(* CODESYS project Test Project V2.project

Project tree, tasks and I/O mapping:
  Device : CODESYS Control Win V3, 3S - Smart Software Solutions GmbH, order no. 305021, version 3.5.7.10
    application Application
      libraries: Standard, * (System)
      task MainTask (cyclic, interval t#500ms, priority 10) calls PLC_PRG
      program PLC_PRG [ST]
  libraries: Standard, 3.5.7.0 (System); SystemTask, 1.3.5.0 (SEL)
  Program/
    Global_Variables/
      global variables Generator_GLV
      global variables Meter_GLV
      global variables Reactive_Bank_GLV
      global variables Run_Time_GLV
    Core Function Blocks/
      function block Circuit_Master [ST]
      function block Power_Control [ST]
      function block Reactive_Control [ST]
      function block Reactive_Bank_Control [ST]
      program Run_Time_Header [ST]
      function block Cap_Bank_Control [ST]
      function block Volt_Var [ST]
      function block Voltage_Control [ST]
    Functions/
      function block PI_Controller [ST]
      function Linearize [ST]
      function PF_to_KVAr [ST]
      Generator_Functions/
        function Generic_Trigger [ST]
        function block Generator_Volt_Var [ST]
        function block Generator_Power_Ramp [ST]
    Interface Blocks/
      function block Reactive_Bank_Interface [ST]
      function block Generic_Generator [ST]
      function block AE_1000NX [ST]
      function block AE_500NX [ST]
      function block SMA_800CP [ST]
      function block SMA_2200CP [ST]
      function block TMEIC_PVL1833 [ST]
      function block Schneider_ConextCore_XC [ST]
      function block SG_1000MX [ST]
*)

// Program/Global_Variables/Generator_GLV
VAR_GLOBAL
	
	// Boolean Reads
	POIV2_Generator_Offline 			: ARRAY[0..99] OF BOOL := [100(0)];
	POIV2_Generator_Fault 				: ARRAY[0..99] OF BOOL := [100(0)];
	POIV2_Generator_DNR					: ARRAY[0..99] OF BOOL := [100(0)];	
	POIV2_Generator_Volt_Var_Protection	: ARRAY[0..99] OF BOOL := [100(0)];
	
	// Boolean Writes
	POIV2_Generator_ON_OFF_CMD 			: ARRAY[0..99] OF BOOL := [100(1)];
	
	//Analog Reads
	POIV2_Circuit_Number 				: ARRAY[0..99] OF REAL := [100(-1)];
	POIV2_Block_Number 					: ARRAY[0..99] OF REAL := [100(-1)];
	POIV2_Generator_Number 				: ARRAY[0..99] OF REAL := [100(-1)];
	POIV2_Generator_KW 					: ARRAY[0..99] OF REAL := [100(1)];
	POIV2_Generator_KVAr 				: ARRAY[0..99] OF REAL := [100(1)];
	POIV2_Generator_PF 					: ARRAY[0..99] OF REAL := [100(1)];
	POIV2_Generator_Max_KW 				: ARRAY[0..99] OF REAL := [100(1)];
	POIV2_Generator_Max_KVAr 			: ARRAY[0..99] OF REAL := [100(1)];
		
	//Analog Writes
	POIV2_Generator_Power_Mode_SP 		: ARRAY[0..99] OF REAL := [100(0)];
	POIV2_Generator_Reactive_Mode_SP 	: ARRAY[0..99] OF REAL := [100(0)];
	POIV2_Generator_Volt_Var_Mode_SP	: ARRAY[0..99] OF REAL := [100(0)];
	POIV2_Generator_PF_SP 				: ARRAY[0..99] OF REAL := [100(1)];
	POIV2_Generator_PF_Ramp_SP 			: ARRAY[0..99] OF REAL := [100(0)];
	POIV2_Generator_KW_Percent_SP		: ARRAY[0..99] OF REAL := [100(100)];
	POIV2_Generator_KW_Ramp_SP 			: ARRAY[0..99] OF REAL := [100(0)];
	POIV2_Generator_KVAr_SP 			: ARRAY[0..99] OF REAL := [100(100)];
	POIV2_Generator_KVAr_Ramp_SP 		: ARRAY[0..99] OF REAL := [100(0)];
	
	//Calculated Analog Reads
	POIV2_Generator_Calculated_KW_Percent_SP 	: ARRAY[0..99] OF REAL := [100(100)];	//Sends feedback from setpoint ramping
	
	POIV2_Power_Redistribution_Mode				: ARRAY[0..99] OF INT := [100(0)]; 
	POIV2_Generator_Overhead_Percent			: ARRAY[0..99] OF REAL := [100(1)];	//Used in Power_Redistribution_Mode
	POIV2_Generator_Surplus_Percent		 		: ARRAY[0..99] OF REAL := [100(1)];	//Used in Power_Redistribution_Mode
	
END_VAR

// Program/Global_Variables/Meter_GLV
VAR_GLOBAL
	// Boolean Reads
	POIV2_Circuit_Breaker_State 	: ARRAY[0..9] OF BOOL := [10(0)];
	POIV2_Circuit_Meter_Offline 	: ARRAY[0..9] OF BOOL := [10(1)];
	                                                          
	//Analog Reads                                            
	POIV2_Circuit_Meter_KW 			: ARRAY[0..9] OF REAL := [10(0)];
	POIV2_Circuit_Meter_KVAr 		: ARRAY[0..9] OF REAL := [10(0)];
	POIV2_Circuit_Meter_PF 			: ARRAY[0..9] OF REAL := [10(1)];
	POIV2_Circuit_Meter_Frequency 	: ARRAY[0..9] OF REAL := [10(0)];
	POIV2_Circuit_Meter_KV 			: ARRAY[0..9] OF REAL := [10(0)];
END_VAR

// Program/Global_Variables/Reactive_Bank_GLV
VAR_GLOBAL


	//Boolean Reads
	POIV2_Cap_Bank_Offline 				: ARRAY[0..9] OF BOOL := [10(0)];
	POIV2_Cap_Bank_Fault 				: ARRAY[0..9] OF BOOL := [10(0)];
	POIV2_Cap_Bank_On	 				: ARRAY[0..9] OF BOOL := [10(0)];
	POIV2_Cap_Bank_Discharging			: ARRAY[0..9] OF BOOL := [10(0)];
	POIV2_Cap_Bank_Switch_Count_Reached	: ARRAY[0..9] OF BOOL := [10(0)];
	
	//Boolean Writes
	POIV2_Cap_Bank_ON_OFF_CMD 			: ARRAY[0..9] OF BOOL := [10(0)];
	POIV2_Cap_Bank_Reset				: ARRAY[0..9] OF BOOL := [10(0)];
	
	
	//Analog Reads
	Reactive_Bank_DNR_Count 			: ARRAY[0..9] OF INT := [10(-1)]; 
	POIV2_Cap_Bank_Circuit_Number 		: ARRAY[0..9] OF INT := [10(-1)];
	POIV2_Cap_Bank_Normalized_KVAr 		: ARRAY[0..9] OF REAL := [10(1000000.0)];
	POIV2_Cap_Bank_Operations_Count 	: ARRAY[0..9] OF REAL ;
	
	
	
	
	
	//Boolean Reads
	POIV2_Reactor_Bank_Offline 				: ARRAY[0..9] OF BOOL := [10(1)];
	POIV2_Reactor_Bank_Fault 				: ARRAY[0..9] OF BOOL := [10(1)];
	POIV2_Reactor_Bank_On	 				: ARRAY[0..9] OF BOOL := [10(0)];
	POIV2_Reactor_Bank_Discharging			: ARRAY[0..9] OF BOOL := [10(0)];
	POIV2_Reactor_Bank_Switch_Count_Reached	: ARRAY[0..9] OF BOOL := [10(0)];
	
	//Boolean Writes
	POIV2_Reactor_Bank_ON_OFF_CMD 			: ARRAY[0..9] OF BOOL := [10(0)];
	POIV2_Reactor_Bank_Reset				: ARRAY[0..9] OF BOOL := [10(0)];
	
	//Analog Reads
	POIV2_Reactor_Bank_Circuit_Number 		: ARRAY[0..9] OF INT := [10(-1)];
	POIV2_Reactor_Bank_Normalized_KVAr 		: ARRAY[0..9] OF REAL := [10(-1000000.0)];
	POIV2_Reactor_Bank_Operations_Count 	: ARRAY[0..9] OF REAL ;
END_VAR

// Program/Global_Variables/Run_Time_GLV
VAR_GLOBAL
	
	//Internal
	
	//{ attribute 'hide' }
	POIV2_Generator_Count	: INT := -1;
	//{ attribute 'hide' }
	POIV2_Reactive_Bank_Count	: INT := -1;
	
	
	
	//{ attribute 'hide' }
	Master_Power_Control_License : BOOL := TRUE;
	//{ attribute 'hide' }
	Master_Reactive_Control_License : BOOL := TRUE;
	
	Power_Control_Disable		: ARRAY[0..10] OF BOOL := [10(1)];
	Reactive_Control_Disable	: ARRAY[0..10] OF BOOL := [10(1)];
	Reactive_Bank_Disable	 	: ARRAY[0..10] OF BOOL := [10(1)];
	Volt_Var_Disable			: ARRAY[0..10] OF BOOL := [10(1)];
	Freq_Watt_Disable			: ARRAY[0..10] OF BOOL := [10(1)]; 
	Voltage_Controller_Disable  : ARRAY[0..10] OF BOOL := [10(1)];
	
	
	//Controller States
	//Controller_States	: ARRAY[0..10] OF BOOL := [10(0)];
	
	//Controller Alarms
	
	
END_VAR

// Device/Application/PLC_PRG
PROGRAM PLC_PRG
VAR 
	Circuit_1_Master : Circuit_Master;
	Circuit_Power_Control : Power_Control;
	Circuit_1_Reactive_Control : Reactive_Control;
	Circuit1_Cap_Control : Cap_Bank_Control;
	
	Circuit1_Circuit_Number			: INT	;
	Circuit1_Breaker_State 			: BOOL	;
	Circuit1_Meter_Offline 			: BOOL	;
	
	Power_Mode : INT;
	counter : INT;
END_VAR

Run_Time_Header();

Circuit_1_Master(
	Circuit_Number	:= 	0,      
	Breaker_State 	:= 	0,      
	Meter_Offline 	:= 	0);   
	
	
	Circuit_Power_Control(
	Circuit_Number:= 0, 
	Disable:= FALSE, 
	Control_Mode:= Power_Mode, 
	Circuit_KW_SP:= 8000, 
	Line_Loss_Modifier:= 1, 
	Circuit_Ramp_Up_Rate:= 60, 
	Circuit_Ramp_Down_Rate:= 60, 
	Generator_Ramp_Rate:= 60, 
	KP:= 0.01, 
	KI:= 1, 
	Run_Cycle:= T#1S);
	
	
	

	Circuit1_Cap_Control(
	Circuit_Number:= 0, 
	Disable:= FALSE, 
	Reset:= FALSE);
	
	
	
	
	
	
	
	
	
	
	
//Test Variables
Circuit_1_Master.Meter_KW 	:= 	Circuit_1_Master.Generators_Gross_KW / 1.05;
Circuit_1_Master.Meter_KVAr := 	Circuit_1_Master.Generators_Gross_KW - 1500 + Circuit1_Cap_Control.Current_Cap_KVAr;
Circuit_1_Master.Meter_PF 	:= LREAL_TO_REAL(Circuit_1_Master.Meter_KW/EXPT(EXPT(Circuit_1_Master.Meter_KW,2)+EXPT(Circuit_1_Master.Meter_KVAr,2),0.5));

FOR counter := 0 TO 99 BY 1 DO
	Generator_GLV.POIV2_Generator_KW[counter] := Generator_GLV.POIV2_Generator_KW_Percent_SP[counter] * 10;
	Generator_GLV.POIV2_Generator_Max_KW[counter] := 1000;
	Generator_GLV.POIV2_Generator_Max_KVAr[counter] := 1000;
	Generator_GLV.POIV2_Generator_KVAr[counter] := linearize(Generator_GLV.POIV2_Generator_PF_SP[counter]) * 1000;
END_FOR

FOR counter := 0 TO 9 BY 1 DO
	Reactive_Bank_GLV.POIV2_Cap_Bank_On[counter] := Reactive_Bank_GLV.POIV2_Cap_Bank_ON_OFF_CMD[counter];
END_FOR

END_PROGRAM

// Program/Core Function Blocks/Run_Time_Header
PROGRAM Run_Time_Header
VAR
	{ attribute 'hide' }
	counter : INT;
	{ attribute 'hide' }
	model : STRING;
	{ attribute 'hide' }
	number : INT;
	{ attribute 'hide' }
	A : BOOL;
	{ attribute 'hide' }
	B : BOOL;
	{ attribute 'hide' }
	C : BOOL;
	{ attribute 'hide' }
	D : BOOL;
END_VAR


Run_Time_GLV.POIV2_Generator_Count 		:= 0;
Run_Time_GLV.POIV2_Reactive_Bank_Count 	:= 0;


Run_Time_GLV.Master_Power_Control_License 		:= TRUE;
Run_Time_GLV.Master_Reactive_Control_License 	:= TRUE;


GET_MOT(Model);
A := FALSE;
B := FALSE;
C := FALSE;
D := FALSE;
Number := 0;
IF(LEFT(Right(Model,2),1) = 'S')THEN
	Number  := STRING_TO_INT(CONCAT('16#',(Right(Model,1))));
	IF(Number > 15)THEN
		Number := 0;
	END_IF
	IF(Number >= 8)THEN
		D := TRUE;
		Number := Number -8;
	END_IF 
	IF(Number >= 4)THEN
		C := TRUE;
		Number := Number - 4;
	END_IF
	IF(Number >= 2)THEN
		B := TRUE;
		Number := Number - 2;
	END_IF
	IF(Number = 1)THEN
		A := TRUE;
		Number := Number - 1;
	END_IF
ELSIF(LEFT(Right(Model,4),2) = 'G1')THEN
	A := TRUE;
	B := TRUE;
ELSE
	A := FALSE;
	B := FALSE;
	C := FALSE;
	D := FALSE;
END_IF


//Run_Time_GLV.Master_Power_Control_License 		:= A;
//Run_Time_GLV.Master_Reactive_Control_License 	:= B;

END_PROGRAM

// Program/Functions/Linearize
FUNCTION Linearize : REAL
VAR_INPUT
	PF : REAL;
END_VAR

IF(PF >= 0)THEN
	Linearize := (1-PF);
ELSE
	Linearize := -1*(1+PF);
END_IF

END_FUNCTION

// Program/Core Function Blocks/Circuit_Master
FUNCTION_BLOCK Circuit_Master
VAR_INPUT
	Circuit_Number			: INT	:= 1;
	Breaker_State 			: BOOL	:= FALSE;
	Meter_Offline 			: BOOL	:= TRUE;
	Meter_KW				: REAL	:= 0;
	Meter_KVAr				: REAL	:= 0;
	Meter_PF				: REAL	:= 1;
	Meter_KV				: REAL	:= 0;
	Meter_Frequency			: REAL	:= 0;
	Generator_Power_Mode	: INT	:= 0; //0 = no power control || 1 = Active Power Limit Control
	Generator_Reactive_Mode	: INT	:= 0; //0 = unity power || 1 = KVAr Control || 2 = Power Factor Control
	Generator_Volt_Var_Mode : INT 	:= 0; //0 = Generators produce VArs even if they trip off to over/under voltage ||1 = Generators produce VArs unill the voltage is too high/low on the output terminals and reduces VArs
END_VAR
VAR_OUTPUT
	Curtail_Licenced					: BOOL;
	PF_Licenced							: BOOL;
	POI_Status 							: INT;
	POI_Alarms 							: INT;
	Generators_In_Control_Loop			: INT;
	Generators_Offline 					: INT;
	Generators_Faulted 					: INT;
	Generators_In_Volt_Var_Protection	: INT;
	Generators_DNR						: INT;
	Generators_Gross_KW 				: REAL;
	Generators_Gross_KVAr 				: REAL;

END_VAR
VAR
	{ attribute 'hide' }
	counter : INT;
END_VAR



// Variable Meter_GLV Writes 			
Meter_GLV.POIV2_Circuit_Breaker_State[Circuit_Number] 	:= Breaker_State; 	
Meter_GLV.POIV2_Circuit_Meter_Offline[Circuit_Number] 	:= Meter_Offline; 	 	
Meter_GLV.POIV2_Circuit_Meter_KW[Circuit_Number] 		:= Meter_KW;
Meter_GLV.POIV2_Circuit_Meter_KVAr[Circuit_Number] 		:= Meter_KVAr;
Meter_GLV.POIV2_Circuit_Meter_PF[Circuit_Number] 		:= Meter_PF;
Meter_GLV.POIV2_Circuit_Meter_Frequency[Circuit_Number] := Meter_Frequency;
Meter_GLV.POIV2_Circuit_Meter_KV[Circuit_Number] 		:= Meter_KV;



// Reset values
Generators_In_Control_Loop	:= 0;
Generators_Offline 			:= 0; 
Generators_Faulted 			:= 0; 
Generators_DNR 				:= 0;
Generators_Gross_KW 		:= 0; 
Generators_Gross_KVAr		:= 0; 

FOR counter := 0 TO 99 BY 1 DO
	IF(Generator_GLV.POIV2_Circuit_Number[counter] = Circuit_Number)THEN
		
		// Variable Generator_GLV Reads
		IF((Generator_GLV.POIV2_Generator_Offline[counter] = 0) AND (Generator_GLV.POIV2_Generator_Fault[counter] = 0))THEN
			Generators_In_Control_Loop 	:= Generators_In_Control_Loop + 1;
		END_IF
		
		Generators_Offline 			:= BOOL_TO_INT(Generator_GLV.POIV2_Generator_Offline[counter])	+ Generators_Offline;
		Generators_Faulted 			:= BOOL_TO_INT(Generator_GLV.POIV2_Generator_Fault[counter]) 	+ Generators_Faulted;
		Generators_DNR 				:= BOOL_TO_INT(Generator_GLV.POIV2_Generator_DNR[counter]) 		+ Generators_DNR;
		Generators_Gross_KW 		:= Generator_GLV.POIV2_Generator_KW[counter] 		+ Generators_Gross_KW;
		Generators_Gross_KVAr		:= Generator_GLV.POIV2_Generator_KVAr[counter] 		+ Generators_Gross_KVAr;
		// Variable Generator_GLV Writes
		Generator_GLV.POIV2_Generator_Power_Mode_SP[counter] 	:= Generator_Power_Mode;
		Generator_GLV.POIV2_Generator_Reactive_Mode_SP[counter] := Generator_Reactive_Mode;
		Generator_GLV.POIV2_Generator_Volt_Var_Mode_SP[counter] := Generator_Volt_Var_Mode;
	END_IF
END_FOR

END_FUNCTION_BLOCK

// Program/Core Function Blocks/Power_Control
FUNCTION_BLOCK Power_Control
VAR_INPUT
	Circuit_Number 			: INT	:= 1;	//Circuit Number for control
	Disable					: BOOL	:= FALSE;	//TRUE fully disables this controller || FALSE enables the controller
	Control_Mode			: INT	:= 0;	//0=Fixed Rate || 1=Dynamic Balance Conservative || 2=Dynamic Balance Moderate || 3=Dynamic Balance Aggressive || 4=PI Control
	Power_Redistribution_Mode: INT	:= 0;   //0=Power Controller sends the same command to all of the Inverters || 1=Inverters Reroute power based on avaliablity  ||Note: Speed Dependant on the feedback time of the end device
	Max_Circuit_KW 			: REAL 	:= 10000; //Maximum AC Power
	Circuit_KW_SP			: REAL	:= 1500;	//KW Circuit Setpoint
	Line_Loss_Modifier		: REAL 	:= 1.02; //
	Circuit_Ramp_Up_Rate	: REAL	:= 10; //KW Per Minute
	Circuit_Ramp_Down_Rate	: REAL	:= 10; //KW Per Minute
	Generator_Ramp_Rate		: REAL	:= 10; //KW Per Minute
	Deadband				: REAL 	:= 10;//Used in PI Control
	KP						: REAL	:= 0.01;//Tuning Parameter for the proportional constant
	KI						: REAL	:= 0.1;//Tuning Parameter for the integral constant
	Run_Cycle				: TIME	:= T#1S;
END_VAR
VAR
	PI_Control : PI_Controller;
	Run_Timer 	: TON;
	Jump_Timer	: TON;
	Offline_Generator_ON_Timer : TON;
	Offline_Generator_OFF_Timer : TON;
	
	counter : INT;
	
	Generators_Count 	: INT;
	Generators_Offline 	: INT;
	Generators_Faulted 	: INT;
	Generators_Gross_KW : REAL;
	Generators_Max_KW 	: REAL;
	Generators_In_Control_Loop : INT;
	Generators_Unknown_Offline_KW 	: REAL;
	Generators_Faulted_KW : REAL;
	
	Final_Circuit_KW_SP : REAL;
	Post_Ramp_Circuit_KW_SP : REAL;
	Offline_Generators_Estimated_Faulted : INT;
	Offline_Generators_KW_Correction : REAL;
	Old_Generators_Offline : INT;
	
	OLD_Generator_KW_Percent : REAL := 100;
	
	OLD_Circuit_KW_SP : REAL := 1000000;
	Ramp_Down_Value : REAL;
	Ramp_Up_Value : REAL;
	
	PI_Control_EN : BOOL := FALSE;
	PI_Control_Offset : REAL;
	
	Generator_KW_Percent : REAL;
	
	Generators_At_SP   : REAL;
	Generator_Overhead : REAL;
	Gross_Generator_Overhead : REAL;
	Generator_Percent_Power_Modif : REAL;
END_VAR




IF(Run_Timer.Q AND NOT(Disable))THEN
	
	//Ramp Rate Logic
	Ramp_Down_Value := LIMIT(0 , (OLD_Circuit_KW_SP - ((Circuit_Ramp_Down_Rate / 60) * TIME_TO_REAL(Run_Cycle)/1000)) , Max_Circuit_KW);
	Ramp_Up_Value   := LIMIT(0 , (OLD_Circuit_KW_SP + ((Circuit_Ramp_Up_Rate / 60) * TIME_TO_REAL(Run_Cycle)/1000)) , Max_Circuit_KW);
	Post_Ramp_Circuit_KW_SP := LIMIT(Ramp_Down_Value , Circuit_KW_SP , Ramp_Up_Value);
	
	// Jump_Logic	
	IF((Circuit_KW_SP < Old_Circuit_KW_SP) AND (Meter_GLV.POIV2_Circuit_Meter_Offline[Circuit_Number] = FALSE) AND Jump_Timer.Q)THEN
		Final_Circuit_KW_SP := LIMIT(Circuit_KW_SP , (Meter_GLV.POIV2_Circuit_Meter_KW[Circuit_Number] * 1.00) , Max_Circuit_KW);
		Jump_Timer(IN := FALSE, PT := T#5M);
	
	ELSE
		Final_Circuit_KW_SP := Post_Ramp_Circuit_KW_SP;
		Jump_Timer(IN := FALSE, PT := T#5M);
	END_IF

	Generators_Count	:= 0;
	Generators_Offline 	:= 0;
	Generators_Faulted 	:= 0;
	Generators_Gross_KW := 0;
	Generators_Max_KW	:= 0;
	Generators_Unknown_Offline_KW 	:= 0;
	Generators_Faulted_KW 			:= 0;
	Generators_In_Control_Loop 		:= 0;

	FOR counter := 0 TO 99 BY 1 DO
		IF(Generator_GLV.POIV2_Circuit_Number[counter] = Circuit_Number)THEN
			Generators_Count 	:= Generators_Count + 1;
			
			// Variable Generator_GLV Reads
			Generators_Offline 	:= BOOL_TO_INT(Generator_GLV.POIV2_Generator_Offline[counter])	+ Generators_Offline;
			Generators_Faulted 	:= BOOL_TO_INT(Generator_GLV.POIV2_Generator_Fault[counter]) 	+ Generators_Faulted;
			Generators_Max_KW	:= Generator_GLV.POIV2_Generator_Max_KW[counter] 				+ Generators_Max_KW;		
						
			IF((Generator_GLV.POIV2_Generator_Offline[counter] = 0) AND (Generator_GLV.POIV2_Generator_Fault[counter] = 0))THEN
				Generators_Gross_KW := Generator_GLV.POIV2_Generator_KW[counter]	+ Generators_Gross_KW;
				Generators_In_Control_Loop 	:= Generators_In_Control_Loop + 1;
				
			END_IF
			
			IF(Generator_GLV.POIV2_Generator_Offline[counter] = 1)THEN
				Generators_Unknown_Offline_KW := Generator_GLV.POIV2_Generator_Max_KW[counter]	+ Generators_Unknown_Offline_KW;
				
			ELSIF(Generator_GLV.POIV2_Generator_Fault[counter] = 1)THEN
				Generators_Faulted_KW := Generator_GLV.POIV2_Generator_Max_KW[counter]	+ Generators_Faulted_KW;
			END_IF			
		END_IF
	END_FOR
	
	
	// Control Mode Logic
	IF((Generators_Max_KW > 0) AND (Generators_In_Control_Loop > 0))THEN
		IF(Control_Mode = 0)THEN
			Generator_KW_Percent	:=	LIMIT(0 , ((Circuit_KW_SP / Generators_Max_KW) * 100) , 100);
		
		ELSIF(Control_Mode = 1)THEN
			Generator_KW_Percent	:=	LIMIT(0 , (((Circuit_KW_SP - Generators_Unknown_Offline_KW) / (Generators_Max_KW - Generators_Unknown_Offline_KW - Generators_Faulted_KW)) * 100) , 100);
		
		ELSIF(Control_Mode = 2)THEN		
		
			IF((Generators_Offline > 0) AND (Meter_GLV.POIV2_Circuit_Meter_Offline[Circuit_Number] = FALSE))THEN
				
				IF((Generators_Offline < OLD_Generators_Offline))THEN
					Offline_Generators_Estimated_Faulted := LIMIT(0 , Offline_Generators_Estimated_Faulted + (Generators_Offline - OLD_Generators_Offline) , Generators_Offline);
					Offline_Generator_ON_Timer(IN := FALSE , PT := T#5M);
					
				ELSIF(Meter_GLV.POIV2_Circuit_Meter_KW[Circuit_Number] > Final_Circuit_KW_SP)THEN
					Offline_Generators_Estimated_Faulted := 0;
					Offline_Generator_ON_Timer(IN := FALSE , PT := T#5M);
				END_IF
					
				IF((Meter_GLV.POIV2_Circuit_Meter_KW[Circuit_Number] < (Final_Circuit_KW_SP - Generators_Unknown_Offline_KW + Offline_Generators_KW_Correction)) AND (Generators_Gross_KW > ((Circuit_KW_SP - Generators_Unknown_Offline_KW + Offline_Generators_KW_Correction)) / 1.05) AND (Generators_Offline <> Offline_Generators_Estimated_Faulted))THEN
					Offline_Generator_ON_Timer(IN := TRUE , PT := T#5M);
				
				ELSE
					Offline_Generator_ON_Timer(IN := FALSE , PT := T#5M);
				END_IF
				
				IF((Meter_GLV.POIV2_Circuit_Meter_KW[Circuit_Number] > (Final_Circuit_KW_SP - Generators_Unknown_Offline_KW + Offline_Generators_KW_Correction)) OR (Generators_Gross_KW < ((Circuit_KW_SP - Generators_Unknown_Offline_KW + Offline_Generators_KW_Correction) / 1.05)) OR (Offline_Generators_Estimated_Faulted > 0))THEN
					Offline_Generator_OFF_Timer(IN := TRUE , PT := T#2M);
					Offline_Generator_ON_Timer(IN := FALSE , PT := T#5M);
					
				ELSE
					Offline_Generator_OFF_Timer(IN := FALSE , PT := T#2M);
				END_IF
				
				IF(Offline_Generator_OFF_Timer.Q)THEN
					Offline_Generators_Estimated_Faulted := LIMIT(0 , Offline_Generators_Estimated_Faulted - 1 , Generators_Offline);
					Offline_Generator_OFF_Timer(IN := FALSE , PT := T#2M);
					Offline_Generator_ON_Timer(IN := FALSE , PT := T#5M);
				END_IF
				
				IF(Offline_Generator_ON_Timer.Q)THEN
					Offline_Generators_Estimated_Faulted := LIMIT(0 , Offline_Generators_Estimated_Faulted + 1 , Generators_Offline);
					Offline_Generator_ON_Timer(IN := FALSE , PT := T#5M);
				END_IF
			
			ELSE
				Offline_Generators_Estimated_Faulted := 0;
			END_IF
			
			IF(Offline_Generators_Estimated_Faulted > 0)THEN
				Offline_Generators_KW_Correction := Generators_Unknown_Offline_KW * (Generators_Offline  / Offline_Generators_Estimated_Faulted);
			ELSE
				Offline_Generators_KW_Correction := 0;			
			END_IF
				
			Old_Generators_Offline := Generators_Offline;
			Generator_KW_Percent	:=	LIMIT(0 , (((Final_Circuit_KW_SP - Generators_Unknown_Offline_KW + Offline_Generators_KW_Correction) / (Generators_Max_KW - Generators_Unknown_Offline_KW - Generators_Faulted_KW + Offline_Generators_KW_Correction)) * 100) , 100);
		
		ELSIF(Control_Mode = 3)THEN
			(*IF((Generators_Gross_KW > (Circuit_KW_SP - Generators_Unknown_Offline_KW ) / 1.02) AND NOT(Meter_GLV.POIV2_Circuit_Meter_Offline[Circuit_Number]) AND (Meter_GLV.POIV2_Circuit_Meter_KW[Circuit_Number] > 1000))THEN
				PI_Control_EN := TRUE;
			ELSIF(Generators_Gross_KW <= (Circuit_KW_SP - Generators_Unknown_Offline_KW ) / 1.05)THEN
				PI_Control_EN := FALSE;
				PI_Control.Reset := TRUE;
				PI_Control_Offset := 0;
			END_IF
			*)
			IF(NOT(Meter_GLV.POIV2_Circuit_Meter_Offline[Circuit_Number]) AND (Meter_GLV.POIV2_Circuit_Meter_KW[Circuit_Number] > (Circuit_KW_SP - (Deadband / 4))))THEN
				//PI_Control_EN := FALSE;
				PI_Control.Reset := TRUE;
				PI_Control_Offset := 0;
			ELSIF(Meter_GLV.POIV2_Circuit_Meter_Offline[Circuit_Number] OR (Generators_Gross_KW / Generators_In_Control_Loop) < (Generator_KW_Percent / 1.05))THEN
				//PI_Control_EN := FALSE;
				PI_Control.Reset := TRUE;
				PI_Control_Offset := 0;
			ELSIF((Generators_Gross_KW / Generators_In_Control_Loop) < (Generator_KW_Percent / 1.01))THEN
				//PI_Control_EN := TRUE;
				PI_Control.Reset := FALSE;
				PI_Control.Hold_Ramp_UP := TRUE;
			ELSE
				//PI_Control_EN := TRUE;
				PI_Control.Reset := FALSE;
				PI_Control.Hold_Ramp_UP := FALSE;
			END_IF
			
			
			//IF(PI_Control_EN)THEN
				PI_Control(
				Reset:= FALSE, 
				Setpoint:= (Circuit_KW_SP - Deadband), 
				Actual_Value:= Meter_GLV.POIV2_Circuit_Meter_KW[Circuit_Number], 
				Output_Ramp_Rate_Up := 0.00166,	// 10 percent per minute		
				Output_Ramp_Rate_Down := 1,
				Output_High_Limit:= 0.2, 
				Output_Low_Limit:= 0, 
				Deadband:= 50, 
				Kp:= KP, 
				Ki:= Ki, 
				Cycle_Time:= Run_Cycle - T#50MS , 
				Output=> PI_Control_Offset);
			//END_IF
		Generator_KW_Percent	:=	LIMIT(0 , ((((Circuit_KW_SP - Generators_Unknown_Offline_KW) / (Generators_Max_KW - Generators_Unknown_Offline_KW - Generators_Faulted_KW)) * 100) * (1 + PI_Control_Offset)) , 100);
		
		ELSIF(Control_Mode = 4)THEN
			PI_Control(
			Reset:= FALSE, 
			Hold_Ramp_Up:= FALSE,
			Setpoint:= Circuit_KW_SP, 
			Actual_Value:= Meter_GLV.POIV2_Circuit_Meter_KW[Circuit_Number], 
			Output_Ramp_Rate_Up := Generator_Ramp_Rate/60,			
			Output_Ramp_Rate_Down := Generator_Ramp_Rate/60,
			Output_High_Limit:= 100, 
			Output_Low_Limit:= 0, 
			Deadband:= Deadband, 
			Kp:= KP, 
			Ki:= Ki, 
			Cycle_Time:= Run_Cycle, 
			Output=> PI_Control_Offset);
			Generator_KW_Percent	:=	LIMIT(0 , PI_Control_Offset , 100);
		
		ELSE
			Generator_KW_Percent	:= Circuit_KW_SP / Max_Circuit_KW;
		END_IF

		
	END_IF
	
	
	//Write to Generator Array
	FOR counter := 0 TO 99 BY 1 DO
		IF(Generator_GLV.POIV2_Circuit_Number[counter] = Circuit_Number)THEN
			// Variable Generator_GLV Write
			Generator_GLV.POIV2_Generator_KW_Percent_SP[counter] := Generator_KW_Percent;
			Generator_GLV.POIV2_Generator_KW_Ramp_SP[counter] := Generator_Ramp_Rate;
		END_IF
	END_FOR
	
	
	OLD_Circuit_KW_SP	:= Circuit_KW_SP;
	OLD_Generator_KW_Percent := Generator_KW_Percent;
	Run_Timer(IN := FALSE, PT := Run_Cycle);
END_IF
Run_Timer(IN := TRUE, PT := Run_Cycle);




// Power Redistribution 
// needs to run every cycle to

IF(Power_Redistribution_Mode = 1)THEN
	//step1 calculate overhead
	Generator_Overhead := 0;
	Generators_At_SP := 0;
	FOR counter := 0 TO 99 BY 1 DO
		IF(Generator_GLV.POIV2_Circuit_Number[counter] = Circuit_Number)THEN
			IF((Generator_GLV.POIV2_Generator_Offline[counter] = 0) AND (Generator_GLV.POIV2_Generator_Fault[counter] = 0))THEN
				Generator_Overhead := LIMIT(0 , Generator_GLV.POIV2_Generator_KW_Percent_SP[counter] - Generator_GLV.POIV2_Generator_Calculated_KW_Percent_SP[counter] , 100);
				Gross_Generator_Overhead := Gross_Generator_Overhead + Generator_Overhead;
				IF(Generator_Overhead = 0)THEN
					Generators_At_SP := Generators_At_SP + 1;
				END_IF			
			END_IF
		END_IF
	END_FOR
	
	//Step2 Calculate the Percentage that the rest of the inverters can increase to
	IF(Generators_At_SP > 0)THEN
		Generator_Percent_Power_Modif := (1+(Gross_Generator_Overhead*(2/Generator_Percent_Power_Modif))/100);
	ELSE
		Generator_Percent_Power_Modif := 1;
	END_IF
	//Step3 Write new values to the inverters
	FOR counter := 0 TO 99 BY 1 DO
		IF(Generator_GLV.POIV2_Circuit_Number[counter] = Circuit_Number)THEN
			// Variable Generator_GLV Write
			Generator_GLV.POIV2_Generator_Overhead_Percent[counter] := Generator_Percent_Power_Modif;
			Generator_GLV.POIV2_Power_Redistribution_Mode[counter] := Power_Redistribution_Mode;
		END_IF
	END_FOR

END_IF

END_FUNCTION_BLOCK

// Program/Functions/PI_Controller
FUNCTION_BLOCK PI_Controller
VAR_INPUT
	Reset 			: BOOL := FALSE;
	Hold_Ramp_UP	: BOOL := FALSE;
	Setpoint		: REAL;
	Actual_Value 	: REAL;
	Output_Ramp_Rate_Up	: REAL;
	Output_Ramp_Rate_Down: REAL;
	Output_High_Limit 	: REAL;
	Output_Low_Limit 	: REAL;
	Deadband 			: REAL;
	Kp 					: REAL;
	Ki 					: REAL;
	Cycle_Time 	: TIME;	
END_VAR
VAR_OUTPUT
	Output : REAL;
END_VAR
VAR
	Cycle_Timer : TON;
	High_Deadband : REAL;
	Low_Deadband : REAL;
	Low_Value : REAL;
	High_Value : REAL;
	Error : REAL;
	Integral : REAL;
	Pre_Ramp_Output : REAL;
	Old_Output : REAL;
END_VAR


IF(Cycle_Timer.Q)THEN
	IF(Reset)THEN
		Integral := 0;
		Old_Output := 0;
		Output := 0;
		Pre_Ramp_Output := 0;
	END_IF

	Low_Deadband := Setpoint  - Deadband;
	High_Deadband := Setpoint + Deadband;
	Error := (Setpoint - Actual_Value) * Kp;
	
	IF((Actual_Value > Low_Deadband) AND (Actual_Value < High_Deadband))THEN
		Error := 0;
	END_IF
	Integral := LIMIT(Output_Low_Limit , (Integral + (error * Ki)) , Output_High_Limit); // Integral Over Run Limit
	
	Pre_Ramp_Output := LIMIT(Output_Low_Limit , (Error + Integral) , Output_High_Limit); 
	
	Low_Value := Old_Output - (Output_Ramp_Rate_Down * TIME_TO_REAL(Cycle_Time)/1000);
	
	IF(Hold_Ramp_UP)THEN
		High_Value := Old_Output;
	ELSE
		High_Value := Old_Output + (Output_Ramp_Rate_Up * TIME_TO_REAL(Cycle_Time)/1000);
	END_IF
	
	Integral := LIMIT(Low_Value , Integral , High_Value);
	Output := LIMIT(Low_Value , Pre_Ramp_Output , High_Value);
	Old_Output := Output;
		
	
	Cycle_Timer(IN := FALSE , PT := Cycle_Time);
END_IF
Cycle_Timer(IN := TRUE , PT := Cycle_Time);

END_FUNCTION_BLOCK

// Program/Core Function Blocks/Reactive_Control
FUNCTION_BLOCK Reactive_Control
VAR_INPUT
	Circuit_Number : INT;
	Disable : BOOL;
	Reactive_Mode : INT; //0 = PF Control ||1 = VAr Control
	Control_Mode : INT; //0 = Open Loop || 1 = Closed Loop PI Control
	Power_Factor_SP : REAL; //Power Factor Setpoint 
	Power_Factor_Ramp_Rate : REAL; // Power Factor Ramp Rate in PF per Second
	KVAr_SP : REAL; // KVAr Control Setpoint
	KVAr_Ramp_Rate : REAL;//KVAr Ramp Rate in KVAr Per Second
	Deadband : REAL;
	Circuit_Lag_Limit : REAL;
	Circuit_Lead_Limit : REAL;
	Generator_Lag_Limit : REAL;
	Generator_Lead_Limit : REAL;
	Kp : REAL;
	Ki : REAL;
	KW_Cutout : REAL;
	Run_Cycle : TIME;
	
END_VAR
VAR
	Run_Timer : TON;
	PF_PI_Control : PI_Controller;
	KVAr_PI_Control : PI_Controller;
	counter : INT;
	Generators_IN_Control_Loop : REAL;
	
	Linearized_Power_Factor_SP : REAL;
	Ramped_Power_Factor_SP : REAL;
	Old_Power_Factor_SP : REAL;
	
	Limited_KVAr_SP : REAL;
	Ramped_KVAr_SP : REAL;
	Old_KVAr_SP : REAL;
	Generator_KVAr_SP : REAL;
	Generator_PF_SP : REAL;
END_VAR


//Status to Run Time 
Run_Time_GLV.Reactive_Control_Disable[Circuit_Number] := Disable;

IF(Run_Timer.Q AND NOT(Disable))THEN
	FOR counter := 0 TO 99 BY 1 DO
		IF(Generator_GLV.POIV2_Circuit_Number[counter] = Circuit_Number)THEN
			// Variable Generator_GLV Reads
			IF((Generator_GLV.POIV2_Generator_Offline[counter] = 0) AND (Generator_GLV.POIV2_Generator_Fault[counter] = 0))THEN
				Generators_In_Control_Loop 	:= Generators_In_Control_Loop + 1;
			END_IF
		END_IF
	END_FOR

	IF((Generators_IN_Control_Loop > 0) AND (Meter_GLV.POIV2_Circuit_Meter_Offline[Circuit_Number] = FALSE))THEN
		IF(Reactive_Mode = 0)THEN
			Generator_KVAr_SP := 0;
			KVAr_PI_Control.Reset := TRUE;
			Linearized_Power_Factor_SP := LIMIT(Linearize(Circuit_Lead_Limit) , Linearize(Power_Factor_SP) , Linearize(Circuit_Lag_Limit));
			Ramped_Power_Factor_SP := LIMIT((Old_Power_Factor_SP - (Power_Factor_Ramp_Rate * TIME_TO_REAL(Run_Cycle)/1000)) , Linearized_Power_Factor_SP , (Old_Power_Factor_SP + (Power_Factor_Ramp_Rate * TIME_TO_REAL(Run_Cycle)/1000)));
			IF(Control_Mode = 0)THEN
				Generator_PF_SP := LIMIT(Linearize(Generator_Lead_Limit) , Ramped_Power_Factor_SP , Linearize(Generator_Lag_Limit));
			ELSIF(Control_Mode =1)THEN
				PF_PI_Control(
				Reset:= FALSE, 
				Hold_Ramp_Up:= FALSE,
				Setpoint:= Ramped_Power_Factor_SP, 
				Actual_Value:= Linearize(Meter_GLV.POIV2_Circuit_Meter_PF[Circuit_Number]), 
				Output_Ramp_Rate_Up := Power_Factor_Ramp_Rate,				
				Output_Ramp_Rate_Down := Power_Factor_Ramp_Rate,
				Output_High_Limit:= Linearize(Generator_Lag_Limit), 
				Output_Low_Limit:= Linearize(Generator_Lead_Limit), 
				Deadband:= Deadband, 
				Kp:= Kp, 
				Ki:= Ki, 
				Cycle_Time:= Run_Cycle, 
				);
				Generator_PF_SP := Linearize(PF_PI_Control.Output);
			END_IF
			Old_Power_Factor_SP := Ramped_Power_Factor_SP;
			
		ELSIF(Reactive_Mode = 1)THEN
			Generator_PF_SP := 1;
			Limited_KVAr_SP := LIMIT(Circuit_Lead_Limit , KVAr_SP , Circuit_Lag_Limit);
			Ramped_KVAr_SP := LIMIT((Old_KVAr_SP - (KVAr_Ramp_Rate  * TIME_TO_REAL(Run_Cycle)/1000)) , Limited_KVAR_SP , (Old_KVAr_SP + (KVAr_Ramp_Rate  * TIME_TO_REAL(Run_Cycle)/1000))); 
			IF(Control_Mode = 0)THEN
				Generator_KVAr_SP := LIMIT(Generator_Lead_Limit , Ramped_KVAr_SP , Generator_Lag_Limit);
			
			ELSIF(Control_Mode = 1)THEN
				KVAr_PI_Control(
				Reset:= FALSE, 
				Hold_Ramp_Up:= FALSE,
				Setpoint:= Ramped_KVAr_SP, 
				Actual_Value:= Meter_GLV.POIV2_Circuit_Meter_KVAr[Circuit_Number], 
				Output_Ramp_Rate_Up:= KVAr_Ramp_Rate, 
				Output_Ramp_Rate_Down:= KVAr_Ramp_Rate, 
				Output_High_Limit:= Generator_Lag_Limit, 
				Output_Low_Limit:= Generator_Lead_Limit, 
				Deadband:= Deadband, 
				Kp:= Kp, 
				Ki:= Ki, 
				Cycle_Time:= Run_Cycle, 
				Output=> Generator_KVAr_SP);
			END_IF
			Old_KVAr_SP := Ramped_KVAr_SP;
		END_IF
	ELSE
		Old_Power_Factor_SP := 1;
		PF_PI_Control.Reset := TRUE;
		Generator_PF_SP := 1;
		Generator_KVAr_SP := 0;
	END_IF
	
	
	
	//Write to Generator Array
	FOR counter := 0 TO 99 BY 1 DO
		IF(Generator_GLV.POIV2_Circuit_Number[counter] = Circuit_Number)THEN
		// Variable Generator_GLV Write
			Generator_GLV.POIV2_Generator_PF[counter] := Generator_PF_SP;
			Generator_GLV.POIV2_Generator_PF_Ramp_SP[counter] := Power_Factor_Ramp_Rate;
			Generator_GLV.POIV2_Generator_KVAr_SP[counter] := Generator_KVAr_SP;
			Generator_GLV.POIV2_Generator_KVAr_Ramp_SP[counter] := KVAr_Ramp_Rate;				
			END_IF
	END_FOR
	Run_Timer(IN := FALSE , PT := Run_Cycle);
END_IF
Run_Timer(IN := TRUE , PT := Run_Cycle);

END_FUNCTION_BLOCK

// Program/Core Function Blocks/Cap_Bank_Control
FUNCTION_BLOCK Cap_Bank_Control
VAR_INPUT
	Circuit_Number : INT;
	Disable : BOOL := FALSE;
	Reset : BOOL := FALSE;
	Control_Mode : INT; //0 = PF Target || 1 = KVAr Target
	Feedback_Mode : INT; //0 = Meter Feedback || 1 = Generator Assist, uses Generator_KVAr
	Generator_KVAr : REAL;//Used in Inverter Assist , Gross Sum of Inverter KVAr 
	Power_Factor_SP : REAL := 1;
	KVAr_SP : REAL := 0;
	Kp : REAL;
	Ki : REAL;
	KVAr_Deadband : REAL := 1000;
	On_Verification_Time : TIME := T#1M;
	KW_Cutout : REAL := 5000;
	KW_Cutout_Threshold : REAL := 1000;
END_VAR
VAR_OUTPUT
	Caps_In_Control_Loop : INT;
	Caps_On	: INT;
	Caps_Faulted : INT;
	Current_Cap_KVAr : REAL; //Current Selected Cap KVAr
END_VAR
VAR
	Time_Over_KVAr : PI_Controller;
	Debounce_Timer : TON;
	counter : INT;
	
	Power_Reset : BOOL := FALSE;
	
	Feedback : REAL;
	Estimated_KVAr_Load : REAL;
	
	//Cap Array Numbers
	Cap_Number_Array : ARRAY[0..3] OF INT := [4(-1)];
	Cap_Array_Index : INT := 0;
	
	//Cap Validity
	Cap_KVAr_Array : ARRAY[0..3] OF REAL := [4(0)];
	//Bubble Sort Variables
	i : INT := 1;
	j : INT := 1;
	flag : INT := 1;
	holding_variable : REAL;
	hold_tracing_variable : INT;
	
	
	Sort_KVAr_Array : ARRAY[0..15] OF REAL := [16(0)];
	
	Deviation_From_Load_Array : ARRAY[0..15] OF REAL := [16(0)]; // Closest Match is index 0
	Tracing_Array  : ARRAY[0..15] OF INT := [16(0)];
	
	Switch : REAL;
	
	Active_Array_Index : INT;
	Binary_Decoder : INT;
END_VAR



//Global Reset
Cap_KVAr_Array[0] := 0;
Cap_KVAr_Array[1] := 0;
Cap_KVAr_Array[2] := 0;
Cap_KVAr_Array[3] := 0;

Tracing_Array[0]  := 0;
Tracing_Array[1]  := 1;
Tracing_Array[2]  := 2;
Tracing_Array[3]  := 3;
Tracing_Array[4]  := 4;
Tracing_Array[5]  := 5;
Tracing_Array[6]  := 6;
Tracing_Array[7]  := 7;
Tracing_Array[8]  := 8;
Tracing_Array[9]  := 9;
Tracing_Array[10] := 10;
Tracing_Array[11] := 11;
Tracing_Array[12] := 12;
Tracing_Array[13] := 13;
Tracing_Array[14] := 14;
Tracing_Array[15] := 15;


IF(NOT(Disable) AND Run_Time_GLV.Master_Reactive_Control_License)THEN
	
	//Power Reset Calcs
	IF(Meter_GLV.POIV2_Circuit_Meter_KW[Circuit_Number] > (KW_Cutout + KW_Cutout_Threshold))THEN
		Power_Reset := FALSE;
	ELSIF(Meter_GLV.POIV2_Circuit_Meter_KW[Circuit_Number] < KW_Cutout)THEN
		Power_Reset := TRUE;
	END_IF

	//For Loop Variable Resets
	Caps_In_Control_Loop := 0;
	Caps_On	:= 0;
	Caps_Faulted := 0;
	Current_Cap_KVAr := 0;
	
	FOR counter := 0 TO 9 BY 1 DO
		IF(Reactive_Bank_GLV.POIV2_Cap_Bank_Circuit_Number[counter] = Circuit_Number)THEN
			
			//Disable Cap Reset
			Reactive_Bank_GLV.POIV2_Cap_Bank_Reset[counter] := FALSE;
			
			//Basic Cap Calculations
			IF(NOT(Reactive_Bank_GLV.POIV2_Cap_Bank_Offline[counter]) AND NOT(Reactive_Bank_GLV.POIV2_Cap_Bank_Fault[counter]))THEN
				Caps_In_Control_Loop := Caps_In_Control_Loop + 1;
			END_IF			
			Caps_On	:= BOOL_TO_INT(Reactive_Bank_GLV.POIV2_Cap_Bank_On[counter]) + Caps_On;
			Caps_Faulted := BOOL_TO_INT(Reactive_Bank_GLV.POIV2_Cap_Bank_Fault[counter]) + Caps_Faulted;
			IF(Reactive_Bank_GLV.POIV2_Cap_Bank_On[counter] AND NOT(Reactive_Bank_GLV.POIV2_Cap_Bank_Offline[counter]) AND NOT(Reactive_Bank_GLV.POIV2_Cap_Bank_Fault[counter]) AND NOT(Reactive_Bank_GLV.POIV2_Cap_Bank_Discharging[counter]) AND NOT(Reactive_Bank_GLV.POIV2_Cap_Bank_Switch_Count_Reached[counter]))THEN
				Current_Cap_KVAr := Reactive_Bank_GLV.POIV2_Cap_Bank_Normalized_KVAr[counter] + Current_Cap_KVAr;
			END_IF
		END_IF	
	
	END_FOR

	IF(Feedback_Mode = 0)THEN
		Feedback := Meter_GLV.POIV2_Circuit_Meter_KVAr[Circuit_Number];
	ELSIF(Feedback_Mode = 1)THEN
		Feedback := Generator_KVAr * -1;
	END_IF
	
	IF(Control_Mode = 0)THEN		
		Estimated_KVAr_Load := PF_to_KVAr(Power_Factor_SP,Circuit_Number);
	ELSIF(Control_Mode = 1)THEN
		Estimated_KVAr_Load := KVAr_SP - Feedback;
	END_IF
	
	// For Loop Resets
	Cap_Number_Array[0] := -1;
	Cap_Number_Array[1] := -1;
	Cap_Number_Array[2] := -1;		
	Cap_Number_Array[3] := -1;
	Cap_Array_Index := 0;
	
	//Find Caps In Circuit
	FOR counter := 0 TO 9 BY 1 DO
		IF(Reactive_Bank_GLV.POIV2_Cap_Bank_Circuit_Number[counter] = Circuit_Number)THEN
			IF(NOT(Reactive_Bank_GLV.POIV2_Cap_Bank_Fault[counter]) OR NOT(Reactive_Bank_GLV.POIV2_Cap_Bank_Offline[counter]) OR NOT(Reactive_Bank_GLV.POIV2_Cap_Bank_Switch_Count_Reached[counter]) OR NOT(Reactive_Bank_GLV.POIV2_Cap_Bank_Discharging[counter]))THEN
				Cap_Number_Array[Cap_Array_Index] := counter;
				Cap_Array_Index := Cap_Array_Index + 1;
			END_IF
		END_IF
	END_FOR
	
	//Dismiss non active caps
	FOR counter := 0 TO 3 BY 1 DO
		IF(Cap_Number_Array[counter] = -1)THEN
			Cap_KVAr_Array[counter] := 987654321;
		ELSE			
			Cap_KVAr_Array[counter] := Reactive_Bank_GLV.POIV2_Cap_Bank_Normalized_KVAr[Cap_Number_Array[counter]];
		END_IF
	END_FOR
	
	

	
	//Binary Combinations
	Sort_KVAr_Array[0]  := 0;																				//0 0 0 0
	Sort_KVAr_Array[1]  := Cap_KVAr_Array[0];																//0 0 0 1
	Sort_KVAr_Array[2]  := Cap_KVAr_Array[1];																//0 0 1 0 
    Sort_KVAr_Array[3]  := Cap_KVAr_Array[0] + Cap_KVAr_Array[1];											//0 0 1 1
    Sort_KVAr_Array[4]  := Cap_KVAr_Array[2];																//0 1 0 0
    Sort_KVAr_Array[5]  := Cap_KVAr_Array[0] + Cap_KVAr_Array[2];											//0 1 0 1
    Sort_KVAr_Array[6]  := Cap_KVAr_Array[1] + Cap_KVAr_Array[2];											//0 1 1 0
    Sort_KVAr_Array[7]  := Cap_KVAr_Array[0] + Cap_KVAr_Array[1] + Cap_KVAr_Array[2];						//0 1 1 1
	Sort_KVAr_Array[8]  := Cap_KVAr_Array[3];																//1 0 0 0
	Sort_KVAr_Array[9]  := Cap_KVAr_Array[0] + Cap_KVAr_Array[3];											//1 0 0 1
	Sort_KVAr_Array[10] := Cap_KVAr_Array[1] + Cap_KVAr_Array[3];											//1 0 1 0 
    Sort_KVAr_Array[11] := Cap_KVAr_Array[0] + Cap_KVAr_Array[1] + Cap_KVAr_Array[3];						//1 0 1 1
    Sort_KVAr_Array[12] := Cap_KVAr_Array[2] + Cap_KVAr_Array[3];											//1 1 0 0
    Sort_KVAr_Array[13] := Cap_KVAr_Array[0] + Cap_KVAr_Array[2] + Cap_KVAr_Array[3];						//1 1 0 1
    Sort_KVAr_Array[14] := Cap_KVAr_Array[1] + Cap_KVAr_Array[2] + Cap_KVAr_Array[3];						//1 1 1 0
    Sort_KVAr_Array[15] := Cap_KVAr_Array[0] + Cap_KVAr_Array[1] + Cap_KVAr_Array[2] + Cap_KVAr_Array[3];	//1 1 1 1
	
	
	
	//Best Match Filter Array Index
	FOR counter := 0 TO 15 BY 1 DO
		Deviation_From_Load_Array[counter] := ABS(Sort_KVAr_Array[counter] - Estimated_KVAr_Load - Current_Cap_KVAr);
	END_FOR
	
	//Bubble Sort
	FOR i := 0 TO 15 BY 1 DO
		FOR j := 0 TO 14 BY 1 DO
			IF(Deviation_From_Load_Array[j + 1] < Deviation_From_Load_Array[j])THEN
				holding_variable := Deviation_From_Load_Array[j + 1];
				hold_tracing_variable := Tracing_Array[j + 1];
				
				Deviation_From_Load_Array[j + 1] := Deviation_From_Load_Array[j ];
				Tracing_Array[j + 1] := Tracing_Array[j];
				
				Deviation_From_Load_Array[j] := holding_variable;
				Tracing_Array[j] := hold_tracing_variable;
			END_IF
		END_FOR
	END_FOR
	
	IF((Estimated_KVAr_Load > (-1 * KVAr_Deadband)) AND (Estimated_KVAr_Load < KVAr_Deadband) OR (ABS(Switch) = 60))THEN
		Time_Over_KVAr.Reset := TRUE;
		//Active_Array_Index := 0;
	ELSE
		Time_Over_KVAr.Reset := FALSE;
	END_IF		
	
	Time_Over_KVAr(
	Hold_Ramp_UP:= FALSE, 
	Setpoint:= Estimated_KVAr_Load, 
	Actual_Value:= 0, 
	Output_Ramp_Rate_Up:= 0.5, 
	Output_Ramp_Rate_Down:= 0.5, 
	Output_High_Limit:= 60, 
	Output_Low_Limit:= -60, 
	Deadband:= KVAr_Deadband, 
	Kp:= Kp, 
	Ki:= Ki, 
	Cycle_Time:= T#0.5S, 
	Output=> Switch);
	
	
	IF(ABS(Switch) = 60)THEN
		Debounce_Timer(IN := TRUE , PT := T#10S);
	ELSE
		Debounce_Timer(PT := T#10S);
	END_IF
	
	IF(Debounce_Timer.Q)THEN
		Debounce_Timer(IN := FALSE , PT := T#10S);
		Active_Array_Index := Tracing_Array[0];
	END_IF
	
	//Reset Prior to writes
	Reactive_Bank_GLV.POIV2_Cap_Bank_ON_OFF_CMD[Cap_Number_Array[0]] := FALSE;
	Reactive_Bank_GLV.POIV2_Cap_Bank_ON_OFF_CMD[Cap_Number_Array[1]] := FALSE;
	Reactive_Bank_GLV.POIV2_Cap_Bank_ON_OFF_CMD[Cap_Number_Array[2]] := FALSE;
	Reactive_Bank_GLV.POIV2_Cap_Bank_ON_OFF_CMD[Cap_Number_Array[3]] := FALSE;
	
	Binary_Decoder := Active_Array_Index;
	IF(Binary_Decoder >= 8)THEN
		Reactive_Bank_GLV.POIV2_Cap_Bank_ON_OFF_CMD[Cap_Number_Array[3]] := TRUE;
		Binary_Decoder := Binary_Decoder -8;
	END_IF 
	IF(Binary_Decoder >= 4)THEN
		Reactive_Bank_GLV.POIV2_Cap_Bank_ON_OFF_CMD[Cap_Number_Array[2]] := TRUE;
		Binary_Decoder := Binary_Decoder - 4;
	END_IF
	IF(Binary_Decoder >= 2)THEN
		Reactive_Bank_GLV.POIV2_Cap_Bank_ON_OFF_CMD[Cap_Number_Array[1]] := TRUE;
		Binary_Decoder := Binary_Decoder - 2;
	END_IF
	IF(Binary_Decoder = 1)THEN
		Reactive_Bank_GLV.POIV2_Cap_Bank_ON_OFF_CMD[Cap_Number_Array[0]] := TRUE;
		Binary_Decoder := Binary_Decoder - 1;
	END_IF

	
	IF(Power_Reset OR RESET)THEN
		FOR counter := 0 TO 9 BY 1 DO
			IF(Reactive_Bank_GLV.POIV2_Cap_Bank_Circuit_Number[counter] = Circuit_Number)THEN
				Reactive_Bank_GLV.POIV2_Cap_Bank_ON_OFF_CMD[counter] := FALSE;
				Reactive_Bank_GLV.POIV2_Cap_Bank_Reset[counter] := TRUE;
				Time_Over_KVAr.Reset := TRUE;
			END_IF
		END_FOR
	END_IF
	
	
END_IF

Reactive_Bank_GLV.Reactive_Bank_DNR_Count[Circuit_Number] := 0;

END_FUNCTION_BLOCK

// Program/Functions/PF_to_KVAr
FUNCTION PF_to_KVAr : REAL
VAR_INPUT
	PF : REAL;
	Circuit_Number : INT;
END_VAR
VAR
END_VAR

// This function converts the Power Factor into a KVAR vector

IF(ABS(PF) = 0)THEN
	PF_to_KVAr := 1;
ELSE
	IF(PF > 0)THEN
		PF_to_KVAr := LREAL_TO_REAL(EXPT((EXPT(Meter_GLV.POIV2_Circuit_Meter_KW[Circuit_Number] / ABS(PF) , 2) - EXPT(Meter_GLV.POIV2_Circuit_Meter_KW[Circuit_Number] , 2)) , 0.5));
	ELSE
		PF_to_KVAr :=  LREAL_TO_REAL(EXPT((EXPT(Meter_GLV.POIV2_Circuit_Meter_KW[Circuit_Number] / ABS(PF) , 2) - EXPT(Meter_GLV.POIV2_Circuit_Meter_KW[Circuit_Number] , 2)) , 0.5) * -1);	
	END_IF
END_IF

END_FUNCTION

// Program/Core Function Blocks/Reactive_Bank_Control
FUNCTION_BLOCK Reactive_Bank_Control
VAR_INPUT
	Circuit_Number : INT;
	System_Time : DATE_AND_TIME; // Resets at midnight
	Disable : BOOL := FALSE;
	Reset : BOOL := FALSE;
	Control_Mode : INT; //0 = PF Target || 1 = KVAr Target
	Feedback_Mode : INT; //0 = Meter Feedback || 1 = Inverter Assist, uses Generator_KVAr
	Generator_KVAr : REAL;//Used in Inverter Assist , Gross Sum of Inverter KVAr 
	Power_Factor_SP : REAL := 1;
	KVAr_SP : REAL := 0;
	On_Verification_Time : TIME := T#5M;
	Min_On_Time : TIME := T#2M;
	KW_Cutout : REAL := 5000;
	KW_Cutout_Threshold : REAL := 1000;
END_VAR
VAR_OUTPUT
	Caps_In_Control_Loop : INT;
	Caps_On	: INT;
	Caps_Faulted : INT;
	
	Reactors_In_Control_Loop : INT;
	Reactors_On	: INT;
	Reactors_Faulted : INT;
END_VAR
VAR_OUTPUT RETAIN
	Cap_Lifetime_Operations : INT;
	Reactor_Lifetime_Operations : INT;	
END_VAR
VAR
	Run_Timer : TON;
	counter : INT;
	
	Power_Reset : BOOL := FALSE;
	
	Feedback : REAL;
	Estimated_KVAr_Load : REAL;
	
	Cap_Runner : INT := 0;
	Cap_Follower : INT := 0;
	Reactor_Runner : INT := 0;
	Reactor_Follower : INT := 0;
	
	Add_Cap : BOOL := FALSE;
	Remove_Cap : BOOL := FALSE;
	Add_Reactor : BOOL := FALSE;
	Remove_Reactor : BOOL := FALSE;
	
	Verification_Timer : TON;
	Min_On_Timer : TON;
	tmp : INT := 0;
END_VAR





IF(NOT(Disable) AND Run_Time_GLV.Master_Reactive_Control_License)THEN
	IF(Run_Timer.Q)THEN
		IF(Meter_GLV.POIV2_Circuit_Meter_KW[Circuit_Number] > (KW_Cutout + KW_Cutout_Threshold))THEN
			Power_Reset := FALSE;
		ELSIF(Meter_GLV.POIV2_Circuit_Meter_KW[Circuit_Number] < KW_Cutout)THEN
			Power_Reset := TRUE;
		END_IF
	
		FOR counter := 0 TO 9 BY 1 DO
			IF(Reactive_Bank_GLV.POIV2_Cap_Bank_Circuit_Number[counter] = Circuit_Number)THEN
				//Disable Cap and Reactor Resets
				Reactive_Bank_GLV.POIV2_Cap_Bank_Reset[counter] := FALSE;				
				Reactive_Bank_GLV.POIV2_Reactor_Bank_Reset[counter] := FALSE;
				
				//Power Limit Reset
				IF(Power_Reset)THEN
					Reactive_Bank_GLV.POIV2_Cap_Bank_ON_OFF_CMD[counter] := FALSE;
					Reactive_Bank_GLV.POIV2_Reactor_Bank_ON_OFF_CMD[counter] := FALSE;	
				END_IF
				
				//Basic Cap Calculations
				IF(NOT(Reactive_Bank_GLV.POIV2_Cap_Bank_Offline[counter]) AND NOT(Reactive_Bank_GLV.POIV2_Cap_Bank_Fault[counter]))THEN
					Caps_In_Control_Loop := Caps_In_Control_Loop + 1;
				END_IF			
				Caps_On	:= BOOL_TO_INT(Reactive_Bank_GLV.POIV2_Cap_Bank_On[counter]) + Caps_On;
				Caps_Faulted := BOOL_TO_INT(Reactive_Bank_GLV.POIV2_Cap_Bank_Fault[counter]) + Caps_Faulted;
			END_IF	
			
			IF(Reactive_Bank_GLV.POIV2_Reactor_Bank_Circuit_Number[counter] = Circuit_Number)THEN
				//Basic Reactor Calculations
				IF(NOT(Reactive_Bank_GLV.POIV2_Reactor_Bank_Offline[counter]) AND NOT(Reactive_Bank_GLV.POIV2_Reactor_Bank_Fault[counter]))THEN
					Reactors_In_Control_Loop := Reactors_In_Control_Loop + 1;
				END_IF
				Reactors_On	:= BOOL_TO_INT(Reactive_Bank_GLV.POIV2_Reactor_Bank_On[counter]) + Reactors_On;
				Reactors_Faulted := BOOL_TO_INT(Reactive_Bank_GLV.POIV2_Reactor_Bank_Fault[counter]) + Reactors_Faulted;
				
			END_IF		
		END_FOR
	
		IF(Feedback_Mode = 0)THEN
			Feedback := Meter_GLV.POIV2_Circuit_Meter_KVAr[Circuit_Number];
		ELSIF(Feedback_Mode = 1)THEN
			Feedback := Generator_KVAr * -1;
		END_IF
		
		IF(Control_Mode = 0)THEN
			Estimated_KVAr_Load := PF_to_KVAr(Power_Factor_SP,Circuit_Number);
		ELSIF(Control_Mode = 1)THEN
			Estimated_KVAr_Load := KVAr_SP - Feedback;
		END_IF
	
	
	
		//Calculate Runners and Followers
		FOR counter := 0 TO 9 BY 1 DO
			//Cap Runner
			IF((Reactive_Bank_GLV.POIV2_Cap_Bank_On[Cap_Runner] AND Reactive_Bank_GLV.POIV2_Cap_Bank_ON_OFF_CMD[Cap_Runner]) OR Reactive_Bank_GLV.POIV2_Cap_Bank_Fault[Cap_Runner] OR Reactive_Bank_GLV.POIV2_Cap_Bank_Offline[Cap_Runner] OR Reactive_Bank_GLV.POIV2_Cap_Bank_Switch_Count_Reached[Cap_Runner] OR Reactive_Bank_GLV.POIV2_Cap_Bank_Discharging[Cap_Runner])THEN
				IF(Cap_Runner >= Caps_In_Control_Loop - 1)THEN
					Cap_Runner := 0;
				ELSE
					Cap_Runner := Cap_Runner + 1;
				END_IF
			END_IF
		
			//Cap Follower
			IF((Reactive_Bank_GLV.POIV2_Cap_Bank_On[Cap_Follower] = FALSE AND Reactive_Bank_GLV.POIV2_Cap_Bank_ON_OFF_CMD[Cap_Follower] = FALSE) OR Reactive_Bank_GLV.POIV2_Cap_Bank_Fault[Cap_Follower] OR Reactive_Bank_GLV.POIV2_Cap_Bank_Offline[Cap_Follower] OR Reactive_Bank_GLV.POIV2_Cap_Bank_Switch_Count_Reached[Cap_Follower] OR Reactive_Bank_GLV.POIV2_Cap_Bank_Discharging[Cap_Follower])THEN
				IF(Cap_Follower >= Caps_In_Control_Loop - 1)THEN
					Cap_Follower := 0;
				ELSE
					Cap_Follower := Cap_Follower + 1;
				END_IF
			END_IF
		
			//Reactor Runner
			IF((Reactive_Bank_GLV.POIV2_Reactor_Bank_On[Reactor_Runner] AND Reactive_Bank_GLV.POIV2_Reactor_Bank_ON_OFF_CMD[Reactor_Runner]) OR Reactive_Bank_GLV.POIV2_Reactor_Bank_Fault[Reactor_Runner] OR Reactive_Bank_GLV.POIV2_Reactor_Bank_Offline[Reactor_Runner] OR Reactive_Bank_GLV.POIV2_Reactor_Bank_Switch_Count_Reached[Reactor_Runner] OR Reactive_Bank_GLV.POIV2_Reactor_Bank_Discharging[Reactor_Runner])THEN
				IF(Reactor_Runner >= Reactors_In_Control_Loop - 1)THEN
					Reactor_Runner := 0;
				ELSE
					Reactor_Runner := Reactor_Runner + 1;
				END_IF
			END_IF
			
			//Reactor Follower
			IF((Reactive_Bank_GLV.POIV2_Reactor_Bank_On[Reactor_Follower] = FALSE AND Reactive_Bank_GLV.POIV2_Reactor_Bank_ON_OFF_CMD[Reactor_Follower] = FALSE) OR Reactive_Bank_GLV.POIV2_Reactor_Bank_Fault[Reactor_Follower] OR Reactive_Bank_GLV.POIV2_Reactor_Bank_Offline[Reactor_Follower] OR Reactive_Bank_GLV.POIV2_Reactor_Bank_Switch_Count_Reached[Reactor_Follower] OR Reactive_Bank_GLV.POIV2_Reactor_Bank_Discharging[Reactor_Follower])THEN
				IF(Reactor_Follower >= Reactors_In_Control_Loop - 1)THEN
					Reactor_Follower := 0;
				ELSE
					Reactor_Follower := Reactor_Follower + 1;
				END_IF
			END_IF
		END_FOR
		
		// Calculation to see if you can add or remove Reactors or Caps
		Add_Cap := 			( 0 < (Estimated_KVAr_Load - Reactive_Bank_GLV.POIV2_Cap_Bank_Normalized_KVAr[Cap_Runner]));
		Remove_Cap := 		( 0 > (Estimated_KVAr_Load + Reactive_Bank_GLV.POIV2_Cap_Bank_Normalized_KVAr[Cap_Follower]));
		Add_Reactor := 		( 0 > (Estimated_KVAr_Load - Reactive_Bank_GLV.POIV2_Reactor_Bank_Normalized_KVAr[Reactor_Runner]));
		Remove_Reactor := 	( 0 < (Estimated_KVAr_Load + Reactive_Bank_GLV.POIV2_Reactor_Bank_Normalized_KVAr[Reactor_Follower]));
		
	
		IF(Reactors_On > 0 OR Caps_On >= Caps_In_Control_Loop OR Caps_In_Control_Loop = 0)THEN
			Add_Cap := FALSE;
		END_IF
		IF(Caps_On > 0 OR Reactors_On >= Reactors_In_Control_Loop OR Reactors_In_Control_Loop = 0)THEN
			Add_Reactor := FALSE;
		END_IF
			
		IF(Caps_On = 0 OR Caps_In_Control_Loop = 0)THEN
			Remove_Cap := FALSE;
		END_IF	
		IF(Reactors_On = 0 OR Reactors_In_Control_Loop = 0)THEN
			Remove_Reactor := FALSE;
		END_IF	
		
	
		//Run Verification Timer to Add Cap or Reactor
		IF((Reactors_On = 0) AND Verification_Timer.Q AND Add_Cap)THEN
			Reactive_Bank_GLV.POIV2_Cap_Bank_ON_OFF_CMD[Cap_Runner] := TRUE;
			Verification_Timer(IN := FALSE, PT := On_Verification_Time);
		END_IF
		IF((Caps_On = 0) AND Verification_Timer.Q AND Add_Reactor)THEN
			Reactive_Bank_GLV.POIV2_Reactor_Bank_ON_OFF_CMD[Reactor_Runner] := TRUE;
			Verification_Timer(IN := FALSE, PT := On_Verification_Time);
		END_IF
			
		//Run Min Time ON to Remove Cap or Reactor
		IF((Caps_On > 0) AND Min_On_Timer.Q AND Remove_Cap)THEN
			Reactive_Bank_GLV.POIV2_Cap_Bank_ON_OFF_CMD[Cap_Follower] := FALSE;
			Min_On_Timer(IN := FALSE, PT := Min_On_Time);
		END_IF
		IF((Reactors_On > 0) AND Min_On_Timer.Q AND Remove_Reactor)THEN
			Reactive_Bank_GLV.POIV2_Reactor_Bank_ON_OFF_CMD[Reactor_Follower] := FALSE;
			Min_On_Timer(IN := FALSE, PT := Min_On_Time);
		END_IF
			
		//Timer Resets
		IF(((Add_Cap =  FALSE AND Add_Reactor = FALSE)) OR Verification_Timer.Q)THEN
			Verification_Timer(IN := FALSE, PT := On_Verification_Time);
		END_IF
		
		IF(((Remove_Cap = FALSE) AND (Remove_Reactor = FALSE)) OR Min_On_Timer.Q)THEN
			Min_On_Timer(IN := FALSE, PT := Min_On_Time);
		END_IF
			
				
		Run_Timer(IN := FALSE , pt := T#10S);
	END_IF
	Run_Timer(IN := TRUE , pt := T#10S);

ELSE
	Verification_Timer(IN := FALSE, PT := On_Verification_Time);
	Min_On_Timer(IN := FALSE, PT := Min_On_Time);
END_IF

//Power Reset Command
IF(Power_Reset OR Reset)THEN
	FOR counter := 0 TO 9 BY 1 DO
		IF(Reactive_Bank_GLV.POIV2_Cap_Bank_Circuit_Number[counter] = Circuit_Number)THEN
			Reactive_Bank_GLV.POIV2_Cap_Bank_ON_OFF_CMD[counter] := FALSE;
			Reactive_Bank_GLV.POIV2_Cap_Bank_Reset[counter] := TRUE;
			Reactive_Bank_GLV.POIV2_Reactor_Bank_ON_OFF_CMD[counter] := FALSE;			
			Reactive_Bank_GLV.POIV2_Reactor_Bank_Reset[counter] := TRUE;
		END_IF
	END_FOR
END_IF




Reactive_Bank_GLV.Reactive_Bank_DNR_Count[Circuit_Number] := 0;

END_FUNCTION_BLOCK

// Program/Interface Blocks/Reactive_Bank_Interface
FUNCTION_BLOCK Reactive_Bank_Interface
VAR_INPUT
	Circuit_Number : INT;
	Offline : BOOL;
	Fault_State : BOOL;
	On_State : BOOL;
	KVAr : REAL;
	Voltage : REAL;
	Rated_Voltage : REAL;
	Discharge_Time : TIME := T#6M;
	Max_Switch_Count : INT := 6;
END_VAR
VAR_OUTPUT
	ON_OFF_CMD : BOOL;
	Trigger : BOOL;
END_VAR
VAR
	Reactive_Unit_Number : INT;
	Discharge_Timer : TON;
	Trigger_Timer : TON;
	Refresh_Timer : TON;
	DNR_Timer : TON;
	Switch_Count : INT;
	Reset : BOOL;
	Normalized_KVAr : REAL;
	Old_Switch_State : BOOL := FALSE;
	Old_Switch_CMD : BOOL := FALSE;
END_VAR

//Initialization
Refresh_Timer(IN := TRUE , PT := T#1M);
Trigger_Timer.PT := T#10S;
Discharge_Timer.PT := Discharge_Time;
DNR_Timer.PT := T#10M;

Reactive_Unit_Number := Run_Time_GLV.POIV2_Reactive_Bank_Count;
Run_Time_GLV.POIV2_Reactive_Bank_Count := Run_Time_GLV.POIV2_Reactive_Bank_Count + 1;

IF(DNR_Timer.Q)THEN
	Fault_State := TRUE;
	Reactive_Bank_GLV.Reactive_Bank_DNR_Count[Circuit_Number] := Reactive_Bank_GLV.Reactive_Bank_DNR_Count[Circuit_Number] + 1;
END_IF


IF(Run_Time_GLV.Master_Reactive_Control_License)THEN
	
	
	//KVAr = 2* pi * farad * (Voltage^2)
	//Normalized KVAr = KVAr/(Rated_KV^2) * (Current_KV^2)
	Normalized_KVAr := KVAr / EXPT(Rated_Voltage , 2) * EXPT(Voltage , 2);
	
	IF(KVAr > 0)THEN //It's a Cap
		Reactive_Bank_GLV.POIV2_Cap_Bank_Offline[Reactive_Unit_Number] 				:= Offline;				
		Reactive_Bank_GLV.POIV2_Cap_Bank_Fault[Reactive_Unit_Number] 				:= Fault_State; 					
		Reactive_Bank_GLV.POIV2_Cap_Bank_On[Reactive_Unit_Number] 					:= On_State;	 					
		Reactive_Bank_GLV.POIV2_Cap_Bank_Discharging[Reactive_Unit_Number] 			:= NOT(Discharge_Timer.Q);			
		Reactive_Bank_GLV.POIV2_Cap_Bank_Switch_Count_Reached[Reactive_Unit_Number]	:= (Switch_Count >= Max_Switch_Count);
		
		ON_OFF_CMD 	:= Reactive_Bank_GLV.POIV2_Cap_Bank_ON_OFF_CMD[Reactive_Unit_Number]; 	
		Reset 		:= Reactive_Bank_GLV.POIV2_Cap_Bank_Reset[Reactive_Unit_Number];
				
		Reactive_Bank_GLV.POIV2_Cap_Bank_Circuit_Number[Reactive_Unit_Number] 	:= Circuit_Number; 
		Reactive_Bank_GLV.POIV2_Cap_Bank_Normalized_KVAr[Reactive_Unit_Number] 	:= Normalized_KVAr;
		Reactive_Bank_GLV.POIV2_Cap_Bank_Operations_Count[Reactive_Unit_Number] := Switch_Count;
	
	ELSE //It's a Shunt Reactor
		Reactive_Bank_GLV.POIV2_Reactor_Bank_Offline[Reactive_Unit_Number] 				:= Offline;				
		Reactive_Bank_GLV.POIV2_Reactor_Bank_Fault[Reactive_Unit_Number] 				:= Fault_State; 					
		Reactive_Bank_GLV.POIV2_Reactor_Bank_On[Reactive_Unit_Number] 					:= On_State;	 					
		Reactive_Bank_GLV.POIV2_Reactor_Bank_Discharging[Reactive_Unit_Number] 			:= NOT(Discharge_Timer.Q);			
		Reactive_Bank_GLV.POIV2_Reactor_Bank_Switch_Count_Reached[Reactive_Unit_Number]	:= (Switch_Count > Max_Switch_Count);
		
		ON_OFF_CMD 	:= Reactive_Bank_GLV.POIV2_Reactor_Bank_ON_OFF_CMD[Reactive_Unit_Number]; 	
		Reset 		:= Reactive_Bank_GLV.POIV2_Reactor_Bank_Reset[Reactive_Unit_Number];
				
		Reactive_Bank_GLV.POIV2_Reactor_Bank_Circuit_Number[Reactive_Unit_Number] 	:= Circuit_Number; 
		Reactive_Bank_GLV.POIV2_Reactor_Bank_Normalized_KVAr[Reactive_Unit_Number] 	:= Normalized_KVAr;
		Reactive_Bank_GLV.POIV2_Reactor_Bank_Operations_Count[Reactive_Unit_Number] := Switch_Count;	
	END_IF
	
	IF(Reset)THEN
		ON_OFF_CMD := FALSE;
		Switch_Count := 0;
	END_IF
	
	IF(Old_Switch_CMD <> ON_OFF_CMD OR Refresh_Timer.Q)THEN
		Trigger := TRUE;
		Trigger_Timer.IN := TRUE;
		Refresh_Timer.IN := FALSE;
	END_IF
	
	IF(Trigger_Timer.Q)THEN
		Trigger := FALSE;
		Trigger_Timer.IN := FALSE;
	END_IF
	
	IF((ON_State <> Old_Switch_State) AND (ON_State = FALSE))THEN // Transition from on to off 
		Discharge_Timer.IN := TRUE;
	END_IF
	
	IF(Discharge_Timer.Q)THEN
		Discharge_Timer.IN := FALSE;
	END_IF
	
	IF(ON_State <> Old_Switch_State)THEN
		Switch_Count := Switch_Count + 1;
	END_IF
	
	IF(ON_State <> ON_OFF_CMD AND NOT(Offline) AND NOT(Fault_State))THEN
		DNR_Timer.IN := TRUE;
	ELSE
		DNR_Timer.IN := FALSE;
	END_IF	
	
	IF(NOT(Run_Time_GLV.Reactive_Bank_Disable[Circuit_Number]))THEN
		Trigger := FALSE;
		Trigger_Timer.IN := FALSE;
		DNR_Timer.IN := FALSE;
		Discharge_Timer.IN := FALSE;		
	END_IF
END_IF

END_FUNCTION_BLOCK

// Program/Interface Blocks/Generic_Generator
FUNCTION_BLOCK Generic_Generator
VAR_INPUT
	Circuit_Number 				: INT;
	Block_Number 				: INT;
	Generator_Number 			: INT;
	
	Offline 					: BOOL;
	Fault_State 				: BOOL;
	On_State 					: BOOL;
	
	KW 							: REAL;
	KVAr 						: REAL;
	Power_Factor 				: REAL;
	Max_KW 						: REAL;
	Max_KVAr 					: REAL;
	
	User_KW_SP 					: REAL := 10000;
END_VAR
VAR_OUTPUT
	KW_Percent_SP 				: REAL;
	KW_SP_Trigger 				: BOOL;
	KW_Percent_Ramp 			: REAL;
	KW_Ramp_Trigger 			: BOOL;

	Power_Factor_SP 			: REAL;
	Power_Factor_Trigger 		: BOOL;
	Power_Factor_Ramp 			: REAL;
	Power_Factor_Ramp_Trigger	: BOOL;
	
	KVAr_Percent_SP 			: REAL;
	KVAr_SP_Trigger 			: BOOL;
	KVAr_Percent_Ramp 			: REAL;
	KVAr_Ramp_Trigger 			: BOOL;	
	
	Power_Mode 					: REAL;
	Reactive_Mode 				: REAL;
	Mode_Trigger				: BOOL;
END_VAR
VAR
	Generator_Unit_Number 		: INT;
	Refresh_Timer 				: TON;
	DNR_Timer 					: TON;
	
	Power_Factor_OOB 			: BOOL;
	KVAr_OOB 					: BOOL;
	Power_Limit_OOB				: BOOL;
END_VAR


Refresh_Timer.PT := T#5M;
DNR_Timer.PT := T#10M;

Generator_Unit_Number := Run_Time_GLV.POIV2_Generator_Count;
Run_Time_GLV.POIV2_Generator_Count := Run_Time_GLV.POIV2_Generator_Count + 1;


IF(Run_Time_GLV.Master_Power_Control_License OR Run_Time_GLV.Master_Reactive_Control_License)THEN
	//Writes to Generator_GLV
	Generator_GLV.POIV2_Generator_Offline[Generator_Unit_Number] 	:= Offline;
	Generator_GLV.POIV2_Generator_Fault[Generator_Unit_Number] 		:= Fault_State; 
	Generator_GLV.POIV2_Generator_DNR[Generator_Unit_Number]		:= DNR_Timer.Q;	
	
	Generator_GLV.POIV2_Circuit_Number[Generator_Unit_Number] 		:=	Circuit_Number;  	
	Generator_GLV.POIV2_Block_Number[Generator_Unit_Number] 		:=	Block_Number;  		
	Generator_GLV.POIV2_Generator_Number[Generator_Unit_Number] 	:=	Generator_Number;  	
	Generator_GLV.POIV2_Generator_KW[Generator_Unit_Number] 		:= 	KW;		
	Generator_GLV.POIV2_Generator_KVAr[Generator_Unit_Number] 		:=	KVAr;  	
	Generator_GLV.POIV2_Generator_PF[Generator_Unit_Number] 		:=	Power_Factor; 		
	Generator_GLV.POIV2_Generator_Max_KW[Generator_Unit_Number] 	:=	Max_KW;  	
	Generator_GLV.POIV2_Generator_Max_KVAr[Generator_Unit_Number] 	:= 	Max_KVAr;

		
	//Generator Writes FROM Generator_GLV
	IF(NOT(Run_Time_GLV.Power_Control_Disable[Circuit_Number]))THEN
		// Triggering and Writes
		KW_SP_Trigger := Generic_Trigger(Generator_GLV.POIV2_Generator_KW_Percent_SP[Generator_Unit_Number],KW_Percent_SP,Refresh_Timer.Q);
		KW_Percent_SP := Generator_GLV.POIV2_Generator_KW_Percent_SP[Generator_Unit_Number];
	
		KW_Ramp_Trigger := Generic_Trigger(Generator_GLV.POIV2_Generator_KW_Ramp_SP[Generator_Unit_Number],KW_Percent_Ramp,Refresh_Timer.Q);
		KW_Percent_Ramp := Generator_GLV.POIV2_Generator_KW_Ramp_SP[Generator_Unit_Number];    
	END_IF      
	
	
	
	
	IF(NOT(Run_Time_GLV.Reactive_Control_Disable[Circuit_Number]))THEN  
		
		// Triggering and Writes
		Power_Factor_Trigger := Generic_Trigger(Generator_GLV.POIV2_Generator_PF_SP[Generator_Unit_Number],Power_Factor_SP,Refresh_Timer.Q);
		Power_Factor_SP := Generator_GLV.POIV2_Generator_PF_SP[Generator_Unit_Number];
		
		Power_Factor_Ramp_Trigger := Generic_Trigger(Generator_GLV.POIV2_Generator_PF_Ramp_SP[Generator_Unit_Number],Power_Factor_Ramp,Refresh_Timer.Q);
		Power_Factor_Ramp := Generator_GLV.POIV2_Generator_PF_Ramp_SP[Generator_Unit_Number]; 
		
		KVAr_SP_Trigger := Generic_Trigger((Generator_GLV.POIV2_Generator_KVAr_SP[Generator_Unit_Number]/Max_KVAr*100),KVAr_Percent_SP,Refresh_Timer.Q);
		KVAr_Percent_SP := (Generator_GLV.POIV2_Generator_KVAr_SP[Generator_Unit_Number]/Max_KVAr*100);
		
		KVAr_Ramp_Trigger := Generic_Trigger(Generator_GLV.POIV2_Generator_KVAr_Ramp_SP[Generator_Unit_Number],KVAr_Percent_Ramp,Refresh_Timer.Q);
		KVAr_Percent_Ramp := Generator_GLV.POIV2_Generator_KVAr_Ramp_SP[Generator_Unit_Number];  
	END_IF
		
	
	IF((Power_Mode <> Generator_GLV.POIV2_Generator_Power_Mode_SP[Generator_Unit_Number]) OR (Reactive_Mode <> Generator_GLV.POIV2_Generator_Reactive_Mode_SP[Generator_Unit_Number]) OR Refresh_Timer.Q)THEN
		Mode_Trigger := TRUE;
	ELSE
		Mode_Trigger := FALSE;
	END_IF		  
	Power_Mode 		:= Generator_GLV.POIV2_Generator_Power_Mode_SP[Generator_Unit_Number];
	Reactive_Mode 	:= Generator_GLV.POIV2_Generator_Reactive_Mode_SP[Generator_Unit_Number];
	
	Refresh_Timer.IN := NOT(Refresh_Timer.Q);
	
	//DNR Logic
	Power_Factor_OOB 	:= (((Linearize(Power_Factor) > Linearize(Power_Factor_SP) + 0.01) OR (Linearize(Power_Factor) < Linearize(Power_Factor_SP) - 0.01)) AND (Generator_GLV.POIV2_Generator_Reactive_Mode_SP[Circuit_Number] = 2));
	KVAr_OOB			:= (((KVAr > Generator_GLV.POIV2_Generator_KVAr_SP[Generator_Unit_Number] + 50) OR (KVAr < Generator_GLV.POIV2_Generator_KVAr_SP[Generator_Unit_Number] - 50)) AND (Generator_GLV.POIV2_Generator_Reactive_Mode_SP[Circuit_Number] = 1));
	Power_Limit_OOB		:= (((KW / Max_KW * 100) > KW_Percent_SP) AND (Generator_GLV.POIV2_Generator_Power_Mode_SP[Circuit_Number] = 1));
	IF((Power_Factor_OOB OR KVAr_OOB OR Power_Limit_OOB) AND ((KW > (Max_KW/4)) AND NOT(Offline) AND NOT(Fault_State)))THEN
		DNR_Timer.IN := TRUE;
	ELSE
		DNR_Timer.IN := FALSE;
	END_IF
		
END_IF

END_FUNCTION_BLOCK

// Program/Functions/Generator_Functions/Generic_Trigger
FUNCTION Generic_Trigger : BOOL
VAR_INPUT
	Input : REAL;
	Feedback : REAL;
	Refresh : BOOL := FALSE;
END_VAR
VAR
END_VAR

IF(Input <> Feedback AND NOT(Refresh))THEN
	Generic_Trigger := TRUE;
ELSE
	Generic_Trigger := FALSE;
END_IF

END_FUNCTION

// Program/Core Function Blocks/Volt_Var
FUNCTION_BLOCK Volt_Var
VAR_INPUT
	Disable : BOOL := TRUE; // True Disables the controller
	Circuit_Number : INT := 0; 
	Power_Factor_SP : REAL := 1; // KVAr_SP needs to be set to 0 before the controller will work to a PF_SP
	KVAr_SP : REAL := 0;
	V1 : REAL := 1.07;
	V2 : REAL := 1.05;
	V3 : REAL := 0.95;
	V4 : REAL := 0.93;
	
	Power_Factor_Lag_Lim : REAL := 0.9;
	Power_Factor_Lead_Lim : REAL := -0.9;	
	
	Hyst_En : BOOL := FALSE;
	Hyst_Threshold : REAL := 0.005;
END_VAR

VAR_OUTPUT
	Power_Factor_Output : REAL;	// Output to the PF controller
	KVAr_Output : REAL; // Output to the VAr controller
	Over_Voltage_Support : BOOL := FALSE; //Indicator the plant is Bucking
	Under_Voltage_Support : BOOL := FALSE; //Indicator the plant is Boosting 
END_VAR
VAR
	Calculated_KVAr_SP : REAL;
	KVAr_Lag_Limit : REAL;
	KVAr_Lead_Limit : REAL;
	Boost_Slope : REAL;
	Buck_Slope : REAL;
END_VAR

//Voltage Bias Written by: Ben Rogowitz	
//This program will bias the POI_PF_Setpoint to allow for partial Voltage Control
//

//Status to Run Time 
Run_Time_GLV.Volt_Var_Disable[Circuit_Number] := Disable;

IF((Disable OR Meter_GLV.POIV2_Circuit_Meter_Offline[Circuit_Number]) OR (Meter_GLV.POIV2_Circuit_Meter_KW[Circuit_Number] < 50))THEN 
	Over_Voltage_Support := FALSE; 
	Under_Voltage_Support := FALSE;
	Power_Factor_Output := Power_Factor_SP;
	KVAr_Output := KVAr_SP;
ELSE
	IF(KVAr_SP = 0)THEN
		Calculated_KVAr_SP := PF_to_KVAr(Power_Factor_SP,Circuit_Number);
	ELSE
		Calculated_KVAr_SP := KVAr_SP;
	END_IF
	
	KVAr_Lag_Limit	:= PF_to_KVAr(Power_Factor_Lag_Lim,Circuit_Number);
	KVAr_Lead_Limit := PF_to_KVAr(Power_Factor_Lead_Lim,Circuit_Number);
	
	Boost_Slope := LIMIT(-999999,(KVAr_Lag_Limit-Calculated_KVAr_SP)/(V1-V2),0);
	Buck_Slope := LIMIT(-999999,(KVAr_Lead_Limit-Calculated_KVAr_SP)/(V4-V3),0);
	
	IF(Hyst_En = FALSE)THEN
		Hyst_Threshold := 0;
	END_IF
	

	//Start Conditions
	IF(Meter_GLV.POIV2_Circuit_Meter_KV[Circuit_Number] < V2)THEN
		Under_Voltage_Support := TRUE;
		Over_Voltage_Support := FALSE;
		
	ELSIF(Meter_GLV.POIV2_Circuit_Meter_KV[Circuit_Number] > V3)THEN
		Under_Voltage_Support := FALSE;
		Over_Voltage_Support := TRUE;
	END_IF
	//End Conditions
	IF(Meter_GLV.POIV2_Circuit_Meter_KV[Circuit_Number] > (V2+Hyst_Threshold))THEN
		Under_Voltage_Support := FALSE;
	END_IF
	IF(Meter_GLV.POIV2_Circuit_Meter_KV[Circuit_Number] < (V3-Hyst_Threshold))THEN
		Over_Voltage_Support := FALSE;
	END_IF

	//Calculate PF Setpoint
	//Boost Condition
	IF(Under_Voltage_Support)THEN
		KVAr_Output := LIMIT(0 , (Meter_GLV.POIV2_Circuit_Meter_KV[circuit_Number]-(V2+Hyst_Threshold))*Boost_Slope , KVAr_Lag_Limit);
		
	//Buck Calculation
	ELSIF(Over_Voltage_Support)THEN
		KVAr_Output := LIMIT(KVAr_Lead_Limit , (Meter_GLV.POIV2_Circuit_Meter_KV[circuit_Number]-(V2+Hyst_Threshold))*Boost_Slope , 0);
	ELSE
		KVAr_Output := LIMIT(KVAr_Lead_Limit , Calculated_KVAr_SP , KVAR_Lag_Limit);
	END_IF
	
	IF(KVAr_Output >= 0)THEN
		Power_Factor_Output := Meter_GLV.POIV2_Circuit_Meter_KW[circuit_Number]/EXPT(EXPT(Meter_GLV.POIV2_Circuit_Meter_KW[circuit_Number],2),EXPT(Meter_GLV.POIV2_Circuit_Meter_KVAr[circuit_Number],2));
	ELSE
		Power_Factor_Output := (Meter_GLV.POIV2_Circuit_Meter_KW[circuit_Number]/EXPT(EXPT(Meter_GLV.POIV2_Circuit_Meter_KW[circuit_Number],2),EXPT(Meter_GLV.POIV2_Circuit_Meter_KVAr[circuit_Number],2))) * -1;			
	END_IF
END_IF

END_FUNCTION_BLOCK

// Program/Interface Blocks/AE_1000NX
FUNCTION_BLOCK AE_1000NX
VAR_INPUT
END_VAR
VAR_OUTPUT
END_VAR
VAR
END_VAR

END_FUNCTION_BLOCK

// Program/Interface Blocks/AE_500NX
FUNCTION_BLOCK AE_500NX
VAR_INPUT
END_VAR
VAR_OUTPUT
END_VAR
VAR
END_VAR

END_FUNCTION_BLOCK

// Program/Interface Blocks/SMA_800CP
FUNCTION_BLOCK SMA_800CP
VAR_INPUT
END_VAR
VAR_OUTPUT
END_VAR
VAR
END_VAR

END_FUNCTION_BLOCK

// Program/Interface Blocks/SMA_2200CP
FUNCTION_BLOCK SMA_2200CP
VAR_INPUT
END_VAR
VAR_OUTPUT
END_VAR
VAR
END_VAR

END_FUNCTION_BLOCK

// Program/Interface Blocks/TMEIC_PVL1833
FUNCTION_BLOCK TMEIC_PVL1833
VAR_INPUT
END_VAR
VAR_OUTPUT
END_VAR
VAR
END_VAR

END_FUNCTION_BLOCK

// Program/Interface Blocks/Schneider_ConextCore_XC
FUNCTION_BLOCK Schneider_ConextCore_XC
VAR_INPUT
END_VAR
VAR_OUTPUT
END_VAR
VAR
END_VAR

END_FUNCTION_BLOCK

// Program/Interface Blocks/SG_1000MX
FUNCTION_BLOCK SG_1000MX
VAR_INPUT
END_VAR
VAR_OUTPUT
END_VAR
VAR
END_VAR

END_FUNCTION_BLOCK

// Program/Functions/Generator_Functions/Generator_Volt_Var
FUNCTION_BLOCK Generator_Volt_Var
VAR_INPUT
	Volt_Var_Mode		: INT := 0;
	Reactive_Mode		: INT := 2;
	Generator_Volts		: REAL := 463;
	Max_PF_Offset		: REAL := 0.2;
	Max_KVAr_Offset		: REAL := 100;
	V1					: REAL := 828; 	//Lowest Voltage where the Generator will still run
	V2					: REAL := 872;	//Highest Voltage where the Generator will still run
	Deadband 			: REAL := 10; //Voltage Offset
	PF_Offset_Array		: ARRAY[1..12] OF REAL := [12(1)];
	KVAr_Offset_Array	: ARRAY[1..12] OF REAL := [12(0)];
END_VAR
VAR_OUTPUT
	In_Volt_Var	: BOOL := 0;
	PF_Offset	: REAL := 0;
	KVAr_Offset	: REAL := 0;
END_VAR
VAR
	PF_Boost_Slope 		: REAL;
	PF_Buck_Slope  		: REAL;
	KVAr_Boost_Slope	: REAL;
	KVAr_Buck_Slope		: REAL;
	
	Under_Voltage_Support 	: BOOL;
	Over_Voltage_Support	: BOOL;
	Timer					: TON;
	PFinst					: REAL;
	KVArinst				: REAL;
	PFHold					: REAL;
	KVArHold				: REAL;
	
	I	: INT;
END_VAR

//Voltage Bias Written by: Ben Rogowitz	
//This program w0Sill bias the POI_PF_Setpoint to allow for partial Voltage Control
//
Timer.PT := T#5S;

//Status to Run Time 
IF(Timer.Q)THEN
	IF(Volt_Var_Mode = 0 OR Reactive_Mode = 0)THEN
		In_Volt_Var	:= 0;
		KVArinst 	:= 0;
		PFinst		:= 0;
	ELSE
	
		PF_Boost_Slope := LIMIT(-999999,(Max_PF_Offset)/(Deadband * -1),0);
		PF_Buck_Slope := LIMIT(-999999,(Max_PF_Offset)/(Deadband * -1),0);
		KVAr_Boost_Slope := LIMIT(-999999,(Max_KVAr_Offset)/(Deadband * -1),0);
		KVAr_Buck_Slope := LIMIT(-999999,(Max_KVAr_Offset)/(Deadband * -1),0);
		
	
		//Start Conditions
		IF(Generator_Volts < (V1 + Deadband))THEN
			Under_Voltage_Support := TRUE;
			Over_Voltage_Support := FALSE;
			
		ELSIF(Generator_Volts > (V2 - Deadband))THEN
			Under_Voltage_Support := FALSE;
			Over_Voltage_Support := TRUE;
		END_IF
		//End Conditions
		IF(Generator_Volts > (V1 + Deadband))THEN
			Under_Voltage_Support := FALSE;
		END_IF
		IF(Generator_Volts < (V2 - Deadband))THEN
			Over_Voltage_Support := FALSE;
		END_IF
		
	
		IF(Under_Voltage_Support)THEN
			KVArinst	:=  LIMIT(0 , (Generator_Volts-(V1 + Deadband))*KVAr_Boost_Slope , Max_KVAr_Offset);
			PFinst		:=  LIMIT(0 , (Generator_Volts-(V1 + Deadband))*PF_Boost_Slope , Max_PF_Offset); 
			In_Volt_Var := TRUE;
		
		ELSIF(Over_Voltage_Support)THEN
			KVArinst 	:=  LIMIT((Max_KVAr_Offset * -1) , (Generator_Volts-(V2 - Deadband))*KVAr_Boost_Slope , 0);
			PFinst		:=  LIMIT((Max_PF_Offset * -1) , (Generator_Volts-(V2 - Deadband))*PF_Boost_Slope , 0); 
			In_Volt_Var := TRUE;
			
		ELSE
			KVArinst 	:= 0;
			PFinst		:= 0;
			In_Volt_Var := FALSE;
			
		END_IF				
	END_IF
	
	//Shift Moving Average Array
	FOR i := 12 TO 2 BY -1 DO
		KVAr_Offset_Array[i] 	:= KVAr_Offset_Array[i-1];
		PF_Offset_Array[i]		:= PF_Offset_Array[i-1];
	END_FOR
	KVAr_Offset_Array[1] 	:= KVArinst;
	PF_Offset_Array[1]		:= PFinst;
	
	//Calcuclate Average from Array
	KVArHold 	:= 0;
	PFHold		:= 0;
	FOR i := 12 TO 2 BY -1 DO
		KVArHold 	:= KVAr_Offset_Array[i] + KVArHold ;
		PFHold		:= PF_Offset_Array[i] + PFHold;
	END_FOR
	PF_Offset	:= (PFHold / 12);
    KVAr_Offset	:= (KVArHold / 12); 
		
	Timer.IN := FALSE;
END_IF
Timer.IN := TRUE;

END_FUNCTION_BLOCK

// Program/Functions/Generator_Functions/Generator_Power_Ramp
FUNCTION_BLOCK Generator_Power_Ramp
VAR_INPUT
	Generator_Number 	: INT;
	Generator_Unable_To_Ramp : BOOL := FALSE; // Use this mode if the inverter can no ramp itself
	Max_Cycle_Time : TIME := T#30s; // this time should be the refresh rate of the inverters + the poll rate of the KW value
END_VAR
VAR_OUTPUT
	Ramped_KW_Percent_SP : REAL;
END_VAR
VAR
	Percent_Power_SP : REAL;
	Redistribution_Percent_Power_SP : REAL;
	Surplus_Percent_Power_SP : REAL;
	Generator_Percent_Power : REAL;
	Ramp_Timer : TON;
	Ramp_Value  : REAL;
	Old_KW : REAL;
END_VAR



Percent_Power_SP := Generator_GLV.POIV2_Generator_KW_Percent_SP[Generator_Number];
Generator_Percent_Power := (Generator_GLV.POIV2_Generator_KW[Generator_Number] / Generator_GLV.POIV2_Generator_Max_KW[Generator_Number] * 100);

IF(Generator_GLV.POIV2_Power_Redistribution_Mode[Generator_Number] = 1)THEN
	Redistribution_Percent_Power_SP := Generator_GLV.POIV2_Generator_Overhead_Percent[Generator_Number];
	Surplus_Percent_Power_SP		:= POIV2_Generator_Surplus_Percent[Generator_Number];
ELSE
	Redistribution_Percent_Power_SP := 0;	
	Surplus_Percent_Power_SP		:= 0;
END_IF

IF(Generator_Unable_To_Ramp)THEN
	Ramp_Timer.PT := Max_Cycle_Time;
	
	IF(Generator_GLV.POIV2_Generator_KW[Generator_Number] <> Old_KW)THEN
		Ramp_Value 	:= (Generator_GLV.POIV2_Generator_KW_Ramp_SP[Generator_Number] * TIME_TO_REAL(Ramp_Timer.ET)/1000);
		
		IF(Generator_Percent_Power <= (Generator_Percent_Power + Redistribution_Percent_Power_SP))THEN
			Ramped_KW_Percent_SP := LIMIT(0 , Generator_GLV.POIV2_Generator_KW[Generator_Number] + Ramp_Value , (Generator_GLV.POIV2_Generator_KW_Percent_SP[Generator_Number] + Generator_GLV.POIV2_Generator_Overhead_Percent[Generator_Number]));
		ELSE
			Ramped_KW_Percent_SP := LIMIT(Generator_Percent_Power,  Generator_GLV.POIV2_Generator_KW[Generator_Number] - Ramp_Value ,  100);
		END_IF
		
		Generator_GLV.POIV2_Generator_Calculated_KW_Percent_SP[Generator_Number] := Ramped_KW_Percent_SP;
		
		Ramp_Timer.IN := FALSE;
	END_IF
	Ramp_Timer.IN := TRUE;

ELSE
	Ramped_KW_Percent_SP := Generator_GLV.POIV2_Generator_KW_Percent_SP[Generator_Number];
	Generator_GLV.POIV2_Generator_Calculated_KW_Percent_SP[Generator_Number] := Ramped_KW_Percent_SP;
END_IF

END_FUNCTION_BLOCK

// Program/Core Function Blocks/Voltage_Control
FUNCTION_BLOCK Voltage_Control
VAR_INPUT	
	Disable : BOOL := TRUE; // True Disables the controller
	Circuit_Number : INT := 0; 
	KVAR_SP : REAL := 0;
	Voltage_SP : REAL;
	POI_Lag_Limit : REAL := 0.95;
	POI_Lead_Limit : REAL := -0.95;
	KP : REAL := 0.002;
	KI : REAL := 0.5;
	KV_Deadband : REAL := 1;
	KVAr_Ramp_Rate : REAL := 1000; //KVAr per Minute
	Cycle_Time : TIME := T#10S;
END_VAR
VAR_OUTPUT
	KVAr_Output : REAL;
END_VAR
VAR
	Voltage_PI : PI_Controller;
	High_KVAr : REAL;
	Low_KVAr : REAL;
END_VAR


IF(Disable OR (Meter_GLV.POIV2_Circuit_Meter_KW[Circuit_Number] < 50))THEN
	KVAr_Output := KVAr_SP;
	
ELSE

	High_KVAr := PF_TO_KVAr(POI_Lag_Limit,Circuit_Number);
	Low_KVAr := PF_TO_KVAr(POI_Lead_Limit,Circuit_Number);
	
	Voltage_PI(
		Reset:= FALSE, 
		Hold_Ramp_UP:= FALSE, 
		Setpoint:= Voltage_SP, 
		Actual_Value:= Meter_GLV.POIV2_Circuit_Meter_KV[Circuit_Number], 
		Output_Ramp_Rate_Up:= KVAr_Ramp_Rate/60, 
		Output_Ramp_Rate_Down:= KVAr_Ramp_Rate/60, 
		Output_High_Limit:= High_KVAr, 
		Output_Low_Limit:= Low_KVAr, 
		Deadband:= KV_Deadband, 
		Kp:= KP, 
		Ki:= KI, 
		Cycle_Time:= Cycle_Time, 
		Output=> KVAr_Output);

END_IF

END_FUNCTION_BLOCK
